	knifeCircumference					:LREAL :=857.65479443007;	(*[mm]*)
	startSyncAngle						:LREAL :=340.0;			(*[°]*)
	endSyncAngle						:LREAL :=20.0;			(*[°]*)
	startAngle							:LREAL :=90.0;			(*[°]*)
	stopAngle							:LREAL :=270.0;			(*[°]*)
	inflectionPoint						:LREAL :=50.0;			(*[%]*)
	numberOfKnives						:INT :=1;
	cutProfileCutOut						:DINT :=0;
	camProfilePhase1					:DINT :=0;
	jerkPhase1							:LREAL :=0.0;			(*[%]*)
	camProfilePhase2					:DINT :=0;
	jerkPhase2							:LREAL :=0.0;			(*[%]*)
	cutProfileCutIn						:DINT :=0;
	distanceToSensor					:LREAL :=0.0;			(*[mm]*)
	firstCutCorrection						:LREAL :=0.0;			(*[mm]*)
	startBacklashOffset					:LREAL :=50.0;			(*[mm]*)
	toStartPosVel						:LREAL :=10.0;			(*[mm/s]*)
	knifeOverspeedStartCut				:LREAL :=0.0;			(*[%]*)
	knifeOverspeedZero					:LREAL :=0.0;			(*[%]*)
	knifeOverspeedEndCut					:LREAL :=0.0;			(*[%]*)
	cpCorrectionMaximum					:LREAL :=0.0;			(*[mm]*)
	cpDeltaToleranceRangePositive			:LREAL :=0.0;			(*[mm]*)
	cpDeltaToleranceRangeNegative			:LREAL :=0.0;			(*[mm]*)
	adjustCutPositionPositiveValue			:LREAL :=0.0;			(*[mm]*)
	trimmCutPositionPositiveValue			:LREAL :=0.0;			(*[mm]*)
	adjustCutPositionNegativeValue			:LREAL :=0.0;			(*[mm]*)
	trimmCutPositionNegativeValue			:LREAL :=0.0;			(*[mm]*)
	cutPositionCorrectionVelocity			:LREAL :=0.0;			(*[mm/s]*)
	cutCorrWait						:INT :=0;
	shiftCorrectionStartPos					:LREAL :=0.0;			(*[%]percentageshiftinformatarea*)
	reStart							:BOOL :=FALSE;
	quickStart							:BOOL :=FALSE;
	formatlengthChangePossible				:BOOL :=FALSE;
	switchCAM							:BOOL :=FALSE;
	measuringEdge						:DINT :=0;
	cutPositionCorrectionOn				:BOOL :=FALSE;
	adjustCutPositionPositive				:BOOL :=FALSE;
	trimmCutPositionPositive				:BOOL :=FALSE;
	adjustCutPositionNegative				:BOOL :=FALSE;
	trimmCutPositionNegative				:BOOL :=FALSE;
	cleanCut							:BOOL :=FALSE;			(*cutwithoutcountingsheets*)
	torquePreControlOn					:BOOL :=FALSE;			(*activationoftorqueprecontrol*)
	totalInertiaOfRotaryKnifeSystem			:LREAL :=0.0;			(*[kgm²]totalinertiaofrotaryknifesystem*)
	torquePreControlMode					:DINT :=0;
	lookAHead							:LREAL :=0.0;			(*[µs]lookaheadtimeinCAM*)
	interruptProduction					:BOOL :=FALSE;
	continueProduction					:BOOL :=FALSE;
	leadingValueCouplingMode				:DINT :=0;
	syncLength							:LREAL :=0.0;			(*[mm]synchronizinglength*)
	extrapolationTime					:LREAL :=0.0;			(*[ms]extrapolationtimeonlyusedbyactualvaluecoupling*)
	constantVelocityAtCut					:BOOL :=FALSE;			(*=synchronousareawithconstantvirtualaxisvelocity,=synchronousareawithactualencodervelocity*)
	startLengthMode						:DINT :=0;
	startLength							:LREAL :=0.0;			(*[mm]*)
	stopLengthMode						:DINT :=0;
	stopLength							:LREAL :=0.0;			(*[mm]*)
	cuttingTorquePreControlOn				:BOOL :=FALSE;
	cuttingTorquePreControlActivePoints		:INT :=0;
	gearInRatioNumerator					:DINT :=0;
	gearInRatioDenominator				:DINT :=0;

END_STRUCT
END_TYPE

// ---- Library/AxisControl/DataTypes/TO_Cam_Struct_PointData.TcDUT
TYPE TO_Cam_Struct_PointData :
STRUCT
	x: LREAL;
	y:LREAL;

END_STRUCT
END_TYPE

// ---- Library/AxisControl/DataTypes/TO_Cam_Struct_SegmentData.TcDUT
TYPE TO_Cam_Struct_SegmentData :
STRUCT

	xmin:LREAL;
	xmax:LREAL;

	a0:LREAL;

	a1:LREAL;

	a2:LREAL;

	a3:LREAL;

	a4:LREAL;

	a5:LREAL;

	a6:LREAL;

	sineAmplitude:LREAL;

	sinePeriod:LREAL;

	sinePhase:LREAL;



END_STRUCT
END_TYPE

// ---- Library/Beckhoff/EL1008/DataTypes/EL1008_DEV_CONFIG.TcDUT
TYPE EL1008_DEV_CONFIG :
STRUCT
    // EN: Enables simulated input values for commissioning and diagnostics.
    // PT: Habilita valores simulados das entradas para comissionamento e diagnóstico.
    enableForce          : BOOL;
    forceDigitalInput_00 : BOOL;
    forceDigitalInput_01 : BOOL;
    forceDigitalInput_02 : BOOL;
    forceDigitalInput_03 : BOOL;
    forceDigitalInput_04 : BOOL;
    forceDigitalInput_05 : BOOL;
    forceDigitalInput_06 : BOOL;
    forceDigitalInput_07 : BOOL;
END_STRUCT
END_TYPE

// ---- Library/Beckhoff/EL1008/DataTypes/EL1008_HWTOPLC_PDOS.TcDUT
TYPE EL1008_HWTOPLC_PDOS :
STRUCT
    // EN: EL1008 EtherCAT input process data.
    // PT: Dados de processo das entradas EtherCAT do EL1008.
    digitalInput_00 AT %I* : BOOL;
    digitalInput_01 AT %I* : BOOL;
    digitalInput_02 AT %I* : BOOL;
    digitalInput_03 AT %I* : BOOL;
    digitalInput_04 AT %I* : BOOL;
    digitalInput_05 AT %I* : BOOL;
    digitalInput_06 AT %I* : BOOL;
    digitalInput_07 AT %I* : BOOL;
END_STRUCT
END_TYPE

// ---- Library/Beckhoff/EL1008/DataTypes/EL1008_PDOS.TcDUT
TYPE EL1008_PDOS :
STRUCT
    HwToPLC : EL1008_HWTOPLC_PDOS;
END_STRUCT
END_TYPE

// ---- Library/Beckhoff/EL1809/DataTypes/EL1809_DEV_CONFIG.TcDUT
TYPE EL1809_DEV_CONFIG :
    STRUCT
       
		enableForce	: BOOL;
		forceDigitalInput_00 : BOOL;
		forceDigitalInput_01 : BOOL;
		forceDigitalInput_02 : BOOL;
		forceDigitalInput_03 : BOOL;
		forceDigitalInput_04 : BOOL;
		forceDigitalInput_05 : BOOL;
		forceDigitalInput_06 : BOOL;
		forceDigitalInput_07 : BOOL;
		forceDigitalInput_08 : BOOL;
		forceDigitalInput_09 : BOOL;
		forceDigitalInput_10 : BOOL;
		forceDigitalInput_11 : BOOL;
		forceDigitalInput_12 : BOOL;
		forceDigitalInput_13 : BOOL;
		forceDigitalInput_14 : BOOL;
		forceDigitalInput_15 : BOOL;


    END_STRUCT
END_TYPE

// ---- Library/Beckhoff/EL1809/DataTypes/EL1809_HWTOPLC_PDOS.TcDUT
TYPE EL1809_HWTOPLC_PDOS :
	STRUCT
		
	
	digitalInput_00 AT %I* : BOOL;
	digitalInput_01 AT %I* : BOOL;
	digitalInput_02 AT %I* : BOOL;
	digitalInput_03 AT %I* : BOOL;
	digitalInput_04 AT %I* : BOOL;
	digitalInput_05 AT %I* : BOOL;
	digitalInput_06 AT %I* : BOOL;
	digitalInput_07 AT %I* : BOOL;
	digitalInput_08 AT %I* : BOOL;
	digitalInput_09 AT %I* : BOOL;
	digitalInput_10 AT %I* : BOOL;
	digitalInput_11 AT %I* : BOOL;
	digitalInput_12 AT %I* : BOOL;
	digitalInput_13 AT %I* : BOOL;
	digitalInput_14 AT %I* : BOOL;
	digitalInput_15 AT %I* : BOOL;


		
	END_STRUCT
END_TYPE

// ---- Library/Beckhoff/EL1809/DataTypes/EL1809_PDOS.TcDUT
TYPE EL1809_PDOS :
	STRUCT
		
		HwToPLC : EL1809_HWTOPLC_PDOS;
		
	END_STRUCT
END_TYPE

// ---- Library/Beckhoff/EL2809/DataTypes/EL2809_DEV_CONFIG.TcDUT
TYPE EL2809_DEV_CONFIG :
    STRUCT
       
		enableForce	: BOOL;
		forceDigitalOutput_00 : BOOL;
		forceDigitalOutput_01 : BOOL;
		forceDigitalOutput_02 : BOOL;
		forceDigitalOutput_03 : BOOL;
		forceDigitalOutput_04 : BOOL;
		forceDigitalOutput_05 : BOOL;
		forceDigitalOutput_06 : BOOL;
		forceDigitalOutput_07 : BOOL;
		forceDigitalOutput_08 : BOOL;
		forceDigitalOutput_09 : BOOL;
		forceDigitalOutput_10 : BOOL;
		forceDigitalOutput_11 : BOOL;
		forceDigitalOutput_12 : BOOL;
		forceDigitalOutput_13 : BOOL;
		forceDigitalOutput_14 : BOOL;
		forceDigitalOutput_15 : BOOL;
			


    END_STRUCT
END_TYPE

// ---- Library/Beckhoff/EL2809/DataTypes/EL2809_PDOS.TcDUT
TYPE EL2809_PDOS :
	STRUCT
		
		PlcToHw : EL2809_PLCTOHW_PDOS;
		
	END_STRUCT
END_TYPE

// ---- Library/Beckhoff/EL2809/DataTypes/EL2809_PLCTOHW_PDOS.TcDUT
TYPE EL2809_PLCTOHW_PDOS :
	STRUCT
		
		digitalOutput_00 AT %Q* : BOOL;
		digitalOutput_01 AT %Q* : BOOL;
		digitalOutput_02 AT %Q* : BOOL;
		digitalOutput_03 AT %Q* : BOOL;
		digitalOutput_04 AT %Q* : BOOL;
		digitalOutput_05 AT %Q* : BOOL;
		digitalOutput_06 AT %Q* : BOOL;
		digitalOutput_07 AT %Q* : BOOL;
		digitalOutput_08 AT %Q* : BOOL;
		digitalOutput_09 AT %Q* : BOOL;
		digitalOutput_10 AT %Q* : BOOL;
		digitalOutput_11 AT %Q* : BOOL;
		digitalOutput_12 AT %Q* : BOOL;
		digitalOutput_13 AT %Q* : BOOL;
		digitalOutput_14 AT %Q* : BOOL;
		digitalOutput_15 AT %Q* : BOOL;

	END_STRUCT
END_TYPE

// ---- Library/Beckhoff/EL3002 - Ai 2 x 10V - 12bit/DataTypes/EL3002_CHANNEL.TcDUT
TYPE EL3002_CHANNEL :
	STRUCT
		
	
	Status 	AT %I* : EL3002_DEV_STATUS;
	Value 	AT %I* : INT;
	
	
	END_STRUCT
END_TYPE

// ---- Library/Beckhoff/EL3002 - Ai 2 x 10V - 12bit/DataTypes/EL3002_DEV_CONFIG.TcDUT
TYPE EL3002_DEV_CONFIG :
    STRUCT
   
        // Setpoint scaling
       	channel1InputLow        : REAL := -32767.0;   // Minimum input value for setpoint		
        channel1InputHigh       : REAL := 32767.0; // Maximum input value for setpoint
        channel1OutputLow       : REAL := -100.0; // Minimum output value for setpoint
        channel1OutputHigh      : REAL := 100.0; // Maximum output value for setpoint
        // Setpoint scaling
       	channe12InputLow        : REAL := -32767.0;   // Minimum input value for setpoint		
        channe12InputHigh       : REAL := 32767.0; // Maximum input value for setpoint
        channe12OutputLow       : REAL := -100.0; // Minimum output value for setpoint
        channe12OutputHigh      : REAL := 100.0; // Maximum output value for setpoint		

    END_STRUCT
END_TYPE

// ---- Library/Beckhoff/EL3002 - Ai 2 x 10V - 12bit/DataTypes/EL3002_DEV_STATUS.TcDUT
TYPE EL3002_DEV_STATUS :
    STRUCT
      
		Underrange : BOOL;
		Overrange : BOOL;
		Limit1 : BOOL;
		Limit2 : BOOL;
		Error : BOOL;
		TxPDOState : BOOL;
		TxPDOToggle : BOOL;
	
    END_STRUCT
END_TYPE

// ---- Library/Beckhoff/EL3002 - Ai 2 x 10V - 12bit/DataTypes/EL3002_HWTOPLC_PDOS.TcDUT
TYPE EL3002_HWTOPLC_PDOS :
	STRUCT
		
	
	Channel1 	AT %I* : EL3002_CHANNEL;
	Channel2 	AT %I* : EL3002_CHANNEL;



	END_STRUCT
END_TYPE

// ---- Library/Beckhoff/EL3002 - Ai 2 x 10V - 12bit/DataTypes/EL3002_PDOS.TcDUT
TYPE EL3002_PDOS :
	STRUCT
		
		HwToPLC : EL3002_HWTOPLC_PDOS;
		
	END_STRUCT
END_TYPE

// ---- Library/Beckhoff/EL4004 - AQ 4 x 0-10V/DataTypes/EL4004_DEV_CONFIG.TcDUT
TYPE EL4004_DEV_CONFIG :
    STRUCT
   
        // Setpoint scaling
       	channel1InputLow        : REAL := 0.0;   // Minimum input value for setpoint		
        channel1InputHigh       : REAL := 100.0; // Maximum input value for setpoint
        channel1OutputLow       : REAL := 0.0; // Minimum output value for setpoint
        channel1OutputHigh      : REAL := 32767.0; // Maximum output value for setpoint

        // Setpoint scaling
       	channel2InputLow        : REAL := 0.0;   // Minimum input value for setpoint		
        channel2InputHigh       : REAL := 100.0; // Maximum input value for setpoint
        channel2OutputLow       : REAL := 0.0; // Minimum output value for setpoint
        channel2OutputHigh      : REAL := 32767.0; // Maximum output value for setpoint

        // Setpoint scaling
       	channel3InputLow        : REAL := 0.0;   // Minimum input value for setpoint		
        channel3InputHigh       : REAL := 100.0; // Maximum input value for setpoint
        channel3OutputLow       : REAL := 0.0; // Minimum output value for setpoint
        channel3OutputHigh      : REAL := 32767.0; // Maximum output value for setpoint

        // Setpoint scaling
       	channel4InputLow        : REAL := 0.0;   // Minimum input value for setpoint		
        channel4InputHigh       : REAL := 100.0; // Maximum input value for setpoint
        channel4OutputLow       : REAL := 0.0; // Minimum output value for setpoint
        channel4OutputHigh      : REAL := 32767.0; // Maximum output value for setpoint


    END_STRUCT
END_TYPE

// ---- Library/Beckhoff/EL4004 - AQ 4 x 0-10V/DataTypes/EL4004_HWTOPLC_PDOS.TcDUT
TYPE EL4004_HWTOPLC_PDOS :
	STRUCT
		
	
	Channel1 	AT %Q* : INT;
	Channel2 	AT %Q* : INT;
	Channel3 	AT %Q* : INT;
	Channel4 	AT %Q* : INT;

	END_STRUCT
END_TYPE

// ---- Library/Beckhoff/EL4004 - AQ 4 x 0-10V/DataTypes/EL4004_PDOS.TcDUT
TYPE EL4004_PDOS :
	STRUCT
		
		HwToPLC : EL4004_HWTOPLC_PDOS;
		
	END_STRUCT
END_TYPE

// ---- Library/Beckhoff/EL5152 -2 x  Encoder Input/DataTypes/EL5152_CONTROL.TcDUT
TYPE EL5152_CONTROL :
STRUCT

		{attribute 'hide'}
		_reserved1 : BIT;
		{attribute 'hide'}
		_reserved2 : BIT;
		Set_counter : BIT;
		{attribute 'hide'}
		_reserved3 : BIT;
		{attribute 'hide'}
		_reserved4 : BIT;
		{attribute 'hide'}
		_reserved5 : BIT;
		{attribute 'hide'}
		_reserved6 : BIT;
		{attribute 'hide'}
		_reserved7 : BIT;
		{attribute 'hide'}
		_reserved8 : USINT;
		
END_STRUCT
END_TYPE

// ---- Library/Beckhoff/EL5152 -2 x  Encoder Input/DataTypes/EL5152_DEV_CONFIG.TcDUT
TYPE EL5152_DEV_CONFIG :
STRUCT

	// Encoder configuration
	encoderPulsePerRevolution	: INT := 2000;      // Number of pulses per revolution (PPR) from the encoder
	encoderScalingFactor	    : REAL := 0.18;      // Position increment per pulse (e.g., 360 mm / 2000 PPR = 0.18 mm/pulse)
	moduloPosition 				: LREAL := 360.0	; // Modulo position range, for example 360.0 

	// Speed calculation
	speedCalculationCycleTime	: TIME := T#300MS;     // Interval at which encoder speed is recalculated

	// Simulation mode
	startSimulation				: BOOL := FALSE;    // Enables encoder simulation mode
	simulatedSpeed				: REAL := 10.0;     // Simulated speed in meters per minute (MPM)

	// Manual position set
	setPosition					: BOOL;             // Trigger to manually set encoder position
	desiredPosition				: LREAL;            // Desired encoder position in millimeters

END_STRUCT
END_TYPE

// ---- Library/Beckhoff/EL5152 -2 x  Encoder Input/DataTypes/EL5152_HWTOPLC.TcDUT
TYPE EL5152_HWTOPLC :
	STRUCT
		
			channel1 : EL5152_HWTOPLC_PDOS;
			channel2 : EL5152_HWTOPLC_PDOS;

	END_STRUCT
END_TYPE

// ---- Library/Beckhoff/EL5152 -2 x  Encoder Input/DataTypes/EL5152_HWTOPLC_PDOS.TcDUT
TYPE EL5152_HWTOPLC_PDOS :
	STRUCT
	
	status												: EL5152_STATUS;	
		{attribute 'hide'}
	_reserved1                                          : UINT;

	CounterValue                              : UDINT; // Current encoder counter value

	END_STRUCT
END_TYPE

// ---- Library/Beckhoff/EL5152 -2 x  Encoder Input/DataTypes/EL5152_PLCTOHW.TcDUT
TYPE EL5152_PLCTOHW :
	STRUCT
		
			channel1 : EL5152_PLCTOHW_PDOS;
			channel2 : EL5152_PLCTOHW_PDOS;

	END_STRUCT
END_TYPE

// ---- Library/Beckhoff/EL5152 -2 x  Encoder Input/DataTypes/EL5152_PLCTOHW_PDOS.TcDUT
TYPE EL5152_PLCTOHW_PDOS :
	STRUCT
		
		control					 : EL5152_CONTROL;
		setCounterValue			 : UDINT; // Sets the encoder counter value
		
	END_STRUCT
END_TYPE

// ---- Library/Beckhoff/EL5152 -2 x  Encoder Input/DataTypes/EL5152_STATUS.TcDUT
TYPE EL5152_STATUS :
STRUCT

		{attribute 'hide'}
		_reserved1 : BIT;
		{attribute 'hide'}
		_reserved2 : BIT;
		Set_counter_done : BIT;
		{attribute 'hide'}
		_reserved3 : BIT;
		{attribute 'hide'}
		_reserved4 : BIT;
		{attribute 'hide'}
		_reserved5 : BIT;
		{attribute 'hide'}
		_reserved6 : BIT;
		Extrapolation_stall : BIT;
		Status_of_input_A : BIT;
		Status_of_input_B : BIT;
		{attribute 'hide'}
		_reserved7 : BIT;
		{attribute 'hide'}
		_reserved8 : BIT;
		{attribute 'hide'}
		_reserved9 : BIT;
		Sync_error : BIT;
		{attribute 'hide'}
		_reserved10 : BIT;
		TxPDO_Toggle : BIT;	

END_STRUCT
END_TYPE

// ---- Library/EL6910 - TwinSAFE PLC/EL6910_ESTOP.TcDUT
TYPE EL6910_ESTOP :
STRUCT
	
	diagnostics : EL6910_ESTOP_DIGNOSTICS;
	status	: EL6910_ESTOP_STATUS;	

END_STRUCT
END_TYPE

// ---- Library/EL6910 - TwinSAFE PLC/EL6910_ESTOP_DIGNOSTICS.TcDUT
TYPE EL6910_ESTOP_DIGNOSTICS :
STRUCT

 	discrepancyErrGroup1       : BOOL; // Discrepancy error input group 1 - BIT00
    discrepancyErrGroup2       : BOOL; // Discrepancy error input group 2 - BIT01
    discrepancyErrGroup3       : BOOL; // Discrepancy error input group 3 - BIT02
    discrepancyErrGroup4       : BOOL; // Discrepancy error input group 4 - BIT03

    edmMonitoringErr1          : BOOL; // EDM monitoring error EDM1 - BIT04
    edmMonitoringErr2          : BOOL; // EDM monitoring error EDM2 - BIT05

    discrepancyErrGroup1_Safe  : BOOL; // Discrepancy error input group 1 with "Safe Inputs after Disc Error" - BIT08
    discrepancyErrGroup2_Safe  : BOOL; // Discrepancy error input group 2 with "Safe Inputs after Disc Error" - BIT09
    discrepancyErrGroup3_Safe  : BOOL; // Discrepancy error input group 3 with "Safe Inputs after Disc Error" - BIT10
    discrepancyErrGroup4_Safe  : BOOL; // Discrepancy error input group 4 with "Safe Inputs after Disc Error" - BIT11

END_STRUCT
END_TYPE

// ---- Library/EL6910 - TwinSAFE PLC/EL6910_ESTOP_STATUS.TcDUT
TYPE EL6910_ESTOP_STATUS :
STRUCT
	
    estopState_RUN        : BOOL; // RUN state 
    estopState_STOP       : BOOL; // STOP state 
    estopState_SAFE       : BOOL; // SAFE state 
    estopState_ERROR      : BOOL; // ERROR state 
    estopState_RESET      : BOOL; // RESET state 
    estopState_START      : BOOL; // START state 
    estopState_DELAYOUT   : BOOL; // DELAYOUT state 
	
END_STRUCT
END_TYPE

// ---- Library/EL6910 - TwinSAFE PLC/EL6910_HWTOPLC_PDOS.TcDUT
TYPE EL6910_HWTOPLC_PDOS :
	STRUCT
			
	EStop1State AT %I* : USINT;
	EStop1Diag 	AT %I* : UINT;
	
	EStop2State AT %I* : USINT;
	EStop2Diag 	AT %I* : UINT;

	EStop3State AT %I* : USINT;
	EStop3Diag 	AT %I* : UINT;

	EStop4State AT %I* : USINT;
	EStop4Diag 	AT %I* : UINT;	
	
	END_STRUCT
END_TYPE

// ---- Library/EL6910 - TwinSAFE PLC/EL6910_PDOS.TcDUT
TYPE EL6910_PDOS :
STRUCT
	
	HwToPLC : EL6910_HWTOPLC_PDOS;
	PlcToHw : EL6910_PLCTOHW_PDOS;			

END_STRUCT
END_TYPE

// ---- Library/EL6910 - TwinSAFE PLC/EL6910_PLCTOHW_PDOS.TcDUT
TYPE EL6910_PLCTOHW_PDOS :
	STRUCT
		
		ErrorAcknowledgement AT %Q* : BOOL;
		safetyReset AT %Q* : BOOL;
	
		Run AT %Q* : BOOL;
		
	END_STRUCT
END_TYPE

// ---- Library/FAS/IO-Link/006B51 - IO-Link Master/DataTypes/_006B51_Channel_State.TcDUT
TYPE _006B51_Channel_State :
STRUCT
	
	inputPin4 	 			: BOOL;
	inputPin2  				: BOOL;
	deviceState  			: BOOL;
	
    state_PortInNoDigitalInput        : BOOL;
    state_PortInNcDigitalInput        : BOOL;
    state_PortInDigitalOutput         : BOOL;
    state_PortInIoLink                : BOOL;

    state_NoDeviceDetected            : BOOL;
    state_IoLinkCommunicationStatus   : BOOL;
    state_InvalidVendorId             : BOOL;
    state_InvalidDeviceId             : BOOL;
    state_InvalidSerialNumber         : BOOL;
    state_InvalidCycleTime            : BOOL;
    state_InvalidProcessDataInLength  : BOOL;
    state_InvalidProcessDataOutLength : BOOL;
    state_InvalidIoLinkVersion        : BOOL;
	
END_STRUCT
END_TYPE

// ---- Library/FAS/IO-Link/006B51 - IO-Link Master/DataTypes/_006B51_HWTOPLC_PDOS.TcDUT
TYPE _006B51_HWTOPLC_PDOS :
STRUCT
	
	inputPin4 	 			: BYTE;
	inputPin2  				: BYTE;
	deviceState  			: BYTE;
	
	ioLinkDeviceState_Port0 : USINT;
	ioLinkDeviceState_Port1 : USINT;
	ioLinkDeviceState_Port2 : USINT;
	ioLinkDeviceState_Port3 : USINT;
	ioLinkDeviceState_Port4 : USINT;
	ioLinkDeviceState_Port5 : USINT;
	ioLinkDeviceState_Port6 : USINT;
	ioLinkDeviceState_Port7 : USINT;
	
END_STRUCT
END_TYPE

// ---- Library/FAS/IO-Link/00BE31 - IP67 16Di or 16Do/DataTypes/_00BE31_HWTOPLC_PDOS.TcDUT
TYPE _00BE31_HWTOPLC_PDOS :
STRUCT
	
	inputByte_0 	 : BYTE;
	inputByte_1  : BYTE;

END_STRUCT
END_TYPE

// ---- Library/FAS/IO-Link/00BE31 - IP67 16Di or 16Do/DataTypes/_00BE31_PLCTOHW_PDOS.TcDUT
TYPE _00BE31_PLCTOHW_PDOS :
STRUCT
	
	outputByte_0 	 : BYTE;
	outputByte_1 	 : BYTE;

END_STRUCT
END_TYPE

// ---- Library/FAS/IO-Link/00BH11 - 16Di or 16Do/DataTypes/_00BH11_HWTOPLC_PDOS.TcDUT
TYPE _00BH11_HWTOPLC_PDOS :
STRUCT
	
	inputByte_0 	 : BYTE;
	inputByte_1  : BYTE;

END_STRUCT
END_TYPE

// ---- Library/FAS/IO-Link/00BH11 - 16Di or 16Do/DataTypes/_00BH11_PLCTOHW_PDOS.TcDUT
TYPE _00BH11_PLCTOHW_PDOS :
STRUCT
	
	outputByte_0 	 : BYTE;
	outputByte_1 	 : BYTE;

END_STRUCT
END_TYPE

// ---- Library/FAS/IO-Link/00BW12 - 16 Solenoid Island/DataTypes/_00BW12_PLCTOHW_PDOS.TcDUT
TYPE _00BW12_PLCTOHW_PDOS :
STRUCT
	
	outputByte_0 	 : BYTE;
	outputByte_1 	 : BYTE;
	outputByte_2 	 : BYTE;
	outputByte_3 	 : BYTE;
	outputByte_4 	 : BYTE;
	outputByte_5 	 : BYTE;
	
END_STRUCT
END_TYPE

// ---- Library/FAS/IO-Link/0AC001 - Analog Input/DataTypes/_0AC001_DEV_CONFIG.TcDUT
TYPE _0AC001_DEV_CONFIG :
STRUCT
	
    // Raw analog input scaling (16-bit: 0..65535)
    analogInputLow   : REAL := 0.0;       // Minimum raw input value
    analogInputHigh  : REAL := 65535.0;   // Maximum raw input value (2 bytes)

    // Engineering-unit output scaling
    analogOutputLow  : REAL := 0.0;       // Engineering value at minimum input
    analogOutputHigh : REAL := 100.0;     // Engineering value at maximum input

END_STRUCT
END_TYPE

// ---- Library/FAS/IO-Link/0AC001 - Analog Input/DataTypes/_0AC001_HWTOPLC_PDOS.TcDUT
TYPE _0AC001_HWTOPLC_PDOS :
STRUCT
	
	inputByte_0 	 : BYTE;
	inputByte_1 	 : BYTE;

END_STRUCT
END_TYPE

// ---- Library/Machine/DryEnd/AutomaticOrderChange/aocConfig_TypeStruct.TcDUT
TYPE aocConfig_TypeStruct :
STRUCT

	automaticOrderChangeSpeed			: REAL	:= 50.0;		(*Automatic order change double facer speed*)

	automaticOrderChangeSpeedMult		: REAL 	:= 2;			(*Automatic order change speed multiplier*)
	rotaryKnifeSpeedMult				: REAL	:= 1;			(*Rotary knife speed multiplier this speed is going to be used to increase the dryend speed*)
	slitterSpeedMult					: REAL	:= 1;			(*slitter speed multiplier this speed is going to be used to reduce the sliiter speed *)

	rampUpTimeSec						: REAL	:= 5.0;		(*Ramp velocity in unit/s, with which the output is changed from a lower value to a higher one.*)
	rampDownTimeSec						: REAL 	:= -5.0;		(*Ramp velocity in unit/s, with which the output is changed from a higher value to a lower one.*)

	aocTimeout							: TIME	:= T#1M;		(*Maximum time to execute the AOC*)
	stackerDischargeDelay				: TIME 	:= T#10S;		(*Small  amout of time that the system  waits after the rotary knife sensor is clear to discharge the stacker*)
	changeSheetLengthTime				: TIME := T#10S;

	
	slitterPaperPresenceDelay					: TIME := T#5S;	
	
	
	speedControlPulseONTime				: TIME := T#1S;
	speedControlPulseOFFTime				: TIME := T#1S;

	
	rotaryShearCutX1MaxTime				: TIME := T#30S;
	measuringWheelClearMaxTime			: TIME := T#30S;	
	slitterClearMaxTime					: TIME := T#30S;	
	rotaryKnifeClearMaxTime				: TIME := T#30S;
	
	

END_STRUCT
END_TYPE

// ---- Library/Machine/DryEnd/AutomaticOrderChange/aocHmiCommands_TypeStruct.TcDUT
TYPE aocHmiCommands_TypeStruct :
STRUCT
	
	aocExecute : BOOL;

END_STRUCT
END_TYPE

// ---- Library/Machine/DryEnd/AutomaticOrderChange/aocHmiStatus_TypeStruct.TcDUT
TYPE aocHmiStatus_TypeStruct :
STRUCT
	
	automaticOrderChangeStatus	: STRING;

END_STRUCT
END_TYPE

// ---- Library/Machine/DryEnd/AutomaticOrderChange/lineControlHmiCommands_TypeStruct.TcDUT
TYPE lineControlHmiCommands_TypeStruct :
STRUCT
	
	speedInc : BOOL;
	speedDec : BOOL;
	speedStop : BOOL;

END_STRUCT
END_TYPE

// ---- Library/Machine/DryEnd/Hmi/hmiAlarms_TypeStruct.TcDUT
TYPE hmiAlarms_TypeStruct :
STRUCT

	slitter : hmiAlarmsSlitter_TypeStruct;
	rotaryKnife : hmiAlarmsRotaryKnife_TypeStruct;
	lowerStacker	: hmiAlarmsSimpleStacker_TypeStruct;
	upperStacker	: hmiAlarmsComplexStacker_TypeStruct;

END_STRUCT
END_TYPE

// ---- Library/Machine/DryEnd/Hmi/hmiCommands_TypeStruct.TcDUT
TYPE hmiCommands_TypeStruct :
STRUCT
	
	orderControl	: orderHmiCommands_TypeStruct;
	lineControl		: lineControlHmiCommands_TypeStruct;	
	slitter1		: slitterCommands_TypeStruct;
	upperKnife		: rotaryKnifeCommands_TypeStruct;
	lowerKnife		: rotaryKnifeCommands_TypeStruct;	
	
	lowerStacker	: hmiCommandsSimpleStacker_TypeStruct;
	upperStacker	: hmiCommandsComplexStacker_TypeStruct;
	
END_STRUCT
END_TYPE

// ---- Library/Machine/DryEnd/Hmi/hmiStatus_TypeStruct.TcDUT
TYPE hmiStatus_TypeStruct :
STRUCT
	alarmActive : BOOL;
		arrKnifeRunningMetersForSharpening		: ARRAY [1..5] OF INT;	(*This array is used to reset the lifetime meters that the knife runs*)
		arrKnifeRunningMetersForLubfrication	: ARRAY [1..5] OF INT;	(*This array is used to reset the lifetime meters that the knife runs*)
		slitter1 : slitterStatus_TypeStruct;
		
		upperKnife								: rotaryKnifeHmiStatus_TypeStruct;
		lowerKnife								: rotaryKnifeHmiStatus_TypeStruct;	
		machineMetrics 							: orderHmiStatus_TypeStruct;
		lowerStacker	: hmiStatusSimpleStacker_TypeStruct;
		upperStacker	: hmiStatusComplexStacker_TypeStruct;

		
END_STRUCT
END_TYPE

// ---- Library/Machine/DryEnd/Hmi/machineConfig_TypeStruct.TcDUT
TYPE machineConfig_TypeStruct :
STRUCT
	
	slitter1 : slitterConfig_TypeStruct;
	upperKnife : rotaryKnifeConfig_TypeStruct;
	lowerKnife	: rotaryKnifeConfig_TypeStruct;	
	automaticOrderChange : aocConfig_TypeStruct;	
	lowerStacker	: SimpleStackerConfig_TypeStruct;
	upperStacker	: ComplexStackerConfig_TypeStruct;

END_STRUCT
END_TYPE

// ---- Library/Machine/DryEnd/Order control/DataTypes/generatedOrderStatusWord_TypeStruct.TcDUT
TYPE generatedOrderStatusWord_TypeStruct :
STRUCT
	

	knifeOutOfRangeArr			: ARRAY [1..5] OF BOOL;
	scorerOutOfRangeArr		: ARRAY [1..8] OF BOOL;


	orderNotOk				: BOOL;	


END_STRUCT
END_TYPE

// ---- Library/Machine/DryEnd/Order control/DataTypes/generatedOrder_TypeStruct.TcDUT
TYPE generatedOrder_TypeStruct :
	STRUCT
		// ========================================================================
		// TOOLING SUMMARY
		// ========================================================================
		numberOfKnifes          : INT;              ///< Total count of active knives in this order
		numberOfScorers         : INT;              ///< Total count of active scorers in this order
		numberOfSheets          : INT;              ///< Total number of sheets in the current production list
		
		// ========================================================================
		// WEB GEOMETRY & CALCULATED WIDTHS [mm]
		// ========================================================================
		order1Width           : REAL;             ///< Calculated width of the Upper level order [mm]
		order2Width        	  : REAL;             ///< Calculated width of the Lower level order [mm]
		orderTotalWidth	      : REAL;             ///< Combined web width (Top + Bottom + Trim) [mm]
		firstKnifePosition      : REAL;             ///< Absolute position of the outermost left knife [mm]
		lastKnifePosition       : REAL;             ///< Absolute position of the outermost right knife [mm]
		
		// ========================================================================
		// KNIFE STATION DATA (Top/Rotary)
		// ========================================================================
		knifeEnabledArr         : ARRAY [1..10] OF BOOL; ///< Tool Enable: TRUE if knife index [x] is required
		knifePositionReferenceArr : ARRAY [1..10] OF REAL; ///< Target position for each knife [mm]
		
		// ========================================================================
		// SCORER STATION DATA (Creasing)
		// ========================================================================
		scorerEnabledArr        : ARRAY [1..20] OF BOOL; ///< Tool Enable: TRUE if scorer index [x] is required
		scorerPositionReferenceArr : ARRAY [1..20] OF REAL; ///< Target position for each scorer [mm]
		// ========================================================================
		// MACHINE STATUS
		// ========================================================================
		statusWord              : generatedOrderStatusWord_TypeStruct; ///< Structured status bits for order validity and errors
				

	END_STRUCT
END_TYPE
		// ========================================================================
		// MACHINE STATUS
		// ========================================================================
//		statusWord              : generatedOrderStatusWord_TypeStruct; ///< Structured status bits for order validity and errors

// ---- Library/Machine/DryEnd/Order control/DataTypes/orderConfig_TypeStruct.TcDUT
TYPE orderConfig_TypeStruct :
STRUCT
	

	automaticReduceMachineSpeed	: BOOL;		(*Reduce machine speed when order finishes*)
	autoStartAOC				: BOOL;		(*Start aoc automatic when the order finishes*)
	
	machineSpeedWhenOrderFinishes	: INT := 50;		(*Machine speed when the machine finishes the order*)
	
	orderFinishingAlertWhenRemainig	: INT := 100;		(*Used to alert the operator when the order is almost finished*)

	measuringWheelDiameter			: REAL := 264.3312;
	
END_STRUCT
END_TYPE

// ---- Library/Machine/DryEnd/Order control/DataTypes/orderHmiCommands_TypeStruct.TcDUT
TYPE orderHmiCommands_TypeStruct :
STRUCT
	
	changeOrder				: BOOL;
	resetUpperLevelCounter	: BOOL;	(*Reset upper level sheet counter*)
	resetLowerLevelCounter	: BOOL;	(*Reset lower level sheet counter*)

END_STRUCT
END_TYPE

// ---- Library/Machine/DryEnd/Order control/DataTypes/orderHmiStatus_TypeStruct.TcDUT
TYPE orderHmiStatus_TypeStruct :
STRUCT
	
	orderFinishing					: BOOL;
	orderFinished					: BOOL;
	linearMetersProduced			: DINT;
	arrMetersPerHour				: ARRAY [0..23] OF INT; (*Meters produced per hour*)
	arrMachineNotRunningTimePerHour	: ARRAY [0..23] OF INT; (*Machine stoped time per hour*)
	arrAverageSpeedPerHour			: ARRAY [0..23] OF INT; (*Machine average speed per hour*)
	machineNotRunningTimeTotal		: INT;
	
END_STRUCT
END_TYPE

// ---- Library/Machine/DryEnd/Order control/DataTypes/orderVariables_TypeStruct.TcDUT
TYPE orderVariables_TypeStruct :
STRUCT
    // ========================================================================
    // CUSTOMER & LOGISTICS DATA
    // ========================================================================
    id                      : DINT;             ///< Unique Order Identification Number
    product                 : STRING;           ///< Product name or internal SKU description
    client                  : STRING;           ///< Customer / Client name
    
    // ========================================================================
    // GEOMETRY & TOOLING CONFIGURATION
    // ========================================================================
    sheetType               : INT := 1;         ///< Scorer config: 0=None, 1=Two Scorers, 2=Four Scorers
    sheetQuantity           : INT := 2;         ///< Number of sheets/outs across the web width
    sheetLength             : INT := 1200;      ///< Cut-off length of each sheet [mm]
    
    // ========================================================================
    // SCORER / CREASER POSITIONS [mm]
    // ========================================================================
    sheetM1                 : INT := 100;       ///< Position of Scorer 1 [mm]
    sheetM2                 : INT := 100;       ///< Position of Scorer 2 [mm]
    sheetM3                 : INT := 100;       ///< Position of Scorer 3 [mm]
    sheetM4                 : INT := 0;         ///< Position of Scorer 4 [mm]
    sheetM5                 : INT := 0;         ///< Position of Scorer 5 [mm]
    
    // ========================================================================
    // PRODUCTION COUNTERS (CUTS)
    // ========================================================================
    numberOfCuts            : DINT;             ///< Total quantity of cuts required for order
    numberOfCutsProduced    : DINT;             ///< Successfully produced cut count
    numberOfCutsRemaining   : DINT;             ///< Calculated: (numberOfCuts - numberOfCutsProduced)
    
    // ========================================================================
    // STACKING & PILE MANAGEMENT
    // ========================================================================
    pileQuantity            : INT := 25;        ///< Target sheet count per finished stack (pile)
    pileQuantityProduced    : INT;              ///< Number of completed piles dispatched
    pileQuantityRemaining   : INT;              ///< Number of piles left to complete the order
    pileCounter             : INT;              ///< Current sheet count in the active pile (resets after pileQuantity)
    
    // ========================================================================
    // QUALITY & WASTE TRACKING
    // ========================================================================
    scrapCounter            : INT;              ///< Count of rejected or wasted sheets
   	counterReset			: BOOL;				///< Counter reset command
	
END_STRUCT
END_TYPE

// ---- Library/Machine/DryEnd/Order control/DataTypes/order_TypeStruct.TcDUT
TYPE order_TypeStruct :
STRUCT
    // ========================================================================
    // DATABASE & TRACKING LOGISTICS
    // ========================================================================
    startedAt               : STRING := '2026-01-11 13:07:00.000'; ///< Timestamp of order initiation
    tableID                 : DINT;                     ///< SQL Database Unique Index/Primary Key
    productionListNumber    : DINT := 92482;            ///< Production Planning System (ERP/MES) ID
    aocRequest      		: BOOL;                     ///< Trigger signal for order transition	
    changeOrderRequest      : BOOL;                     ///< Trigger signal for order transition
    saveSQLFinished         : BOOL;                     ///< Feedback: Database write operation successful
    saveSQLTimeOut          : BOOL;                     ///< Feedback: Database connection/write failure
   	plcWatchDog				: BOOL;
 
    // ========================================================================
    // BOARD SPECIFICATIONS (GRADE & COMPOSITION)
    // ========================================================================
    paperComposition        : STRING := 'KF3MF3K/BC 670G/M²'; ///< Board grade and total weight description
    fluteType               : STRING := 'BC';           ///< Corrugation profile (e.g., Single/Double Wall)
    paperWidth              : INT := 1810;              ///< Raw paper web width [mm]
    
    // ========================================================================
    // PAPER LAYER DEFINITIONS (LINERS & MEDIUMS)
    // ========================================================================
    paper1                  : STRING := 'KRAFT-90';     ///< Layer 1: Top Liner (Face)
    paper2                  : STRING := 'MIOLO F-130';  ///< Layer 2: Fluting 1 (Medium)
    paper3                  : STRING := 'MIOLO-90';     ///< Layer 3: Center Liner
    paper4                  : STRING := 'MIOLO-90';     ///< Layer 4: Fluting 2 (Medium)
    paper5                  : STRING := 'MIOLO-90';     ///< Layer 5: Bottom Liner (Back)
    
    // ========================================================================
    // PRODUCTION METRICS & KPI TRACKING
    // ========================================================================
    lineSpeed               : REAL;                     ///< Current machine velocity [m/min]
    linearMeters            : REAL := 2208.0;           ///< Total target length for the order [m]
    linearMetersProduced    : REAL;                     ///< Actual quantity processed [m]
    linearMetersRemaining   : REAL;                     ///< Calculated distance until completion [m]
    
    // ========================================================================
    // TOOLING & EXECUTION CONTROL
    // ========================================================================
    scorerHeightMM          : REAL := 0.5;              ///< Target penetration depth for slitter-scorer tools [mm]
    levelSelector           : E_LevelSelector := 1;     ///< Active Level: 1=Upper, 2=Lower, 3=Both
    invertOrderLevel        : BOOL;                     ///< Flag to swap logic between physical machine levels
    invertOrderSide         : BOOL;                     ///< Flag to swap order data between Order 1 and Order 2
 
    // ========================================================================
    // CHILD STRUCTURES (DETAILED PARAMETERS)
    // ========================================================================
    order1                  : OrderVariables_TypeStruct; ///< Config parameters for Upper Knife station
    order2                  : OrderVariables_TypeStruct; ///< Config parameters for Lower Knife station
    generatedOrder          : GeneratedOrder_TypeStruct; ///< Resultant set calculated for machine execution
    
END_STRUCT
END_TYPE

// ---- Library/Machine/DryEnd/Order control/DataTypes/sheetTypeEnum.TcDUT
(*
This enumerator is used to define the type of sheet that is going to be
produced by the machine
*)

TYPE sheetTypeEnum:
 (
	SHEET_WITH_NO_SCORER,		(* Sheet with no scoring marks*)
	SHEET_WITH_TWO_SCORER,		(* Sheet with two socoring marks *)
	SHEET_WITH_FOUR_SCORER		(*Sheet with four socoring marks*)

 );
END_TYPE

// ---- Library/Machine/Rotary knife/Config/rotaryKnifeConfig_TypeStruct.TcDUT
(*
TYPE rotaryKnifeConfig_TypeStruct :
STRUCT
	
	infeedRollSpeedOffset	: REAL	:= 1.1;
	outfeedRollSpeedOffset	: REAL	:= 1.2;
	minLineSpeed			: REAL := 20.0;
	
	switchEncoderDelay			: TIME := T#30S;
	speedCurve				    : ARRAY [1..10] OF rotaryKnifeSpeedCurve_TypeConfig;

	lengthAdjustment			: INT;
	
END_STRUCT
END_TYPE 
*)
TYPE rotaryKnifeConfig_TypeStruct :
STRUCT
    
    // --- Roll Speed Ratios ---
    infeedRollSpeedOffset   : REAL := 1.1;  // Multiplier for infeed roll speed relative to line speed (e.g., 1.1 = 10% draw)
    outfeedRollSpeedOffset  : REAL := 1.2;  // Multiplier for outfeed roll speed to maintain tension/gap after cut
    
    // --- Operational Limits ---
    minLineSpeed            : REAL := 20.0; // Minimum line speed (e.g., m/min) to allow automatic operation
    
    // --- Geometry & Logic ---
    enableSyncDiameter      : BOOL;         // TRUE: Use synchronous cutting if sheet length < Knife Circumference (π * D)
    knifeDiameter           : REAL := 262.670; // Physical diameter of the knife cylinder (mm)
    knifeDiameterFactor           	: REAL := 1.0; // Physical diameter of the knife cylinder (mm)
    
	
    // --- Timing & Profiles ---
    switchEncoderDelay      : TIME := T#30S; // Delay/filter time when toggling between feedback encoders
    speedCurve              : ARRAY [1..10] OF rotaryKnifeSpeedCurve_TypeConfig; // CAM or velocity profiles for different materials/speeds

    // --- Fine Tuning ---
    lengthAdjustment        : INT;          // Global position offset (pulses or tenths of mm) to trim cut accuracy
    
END_STRUCT
END_TYPE

// ---- Library/Machine/Rotary knife/Config/rotaryKnifeHmiStatus_TypeStruct.TcDUT
TYPE rotaryKnifeHmiStatus_TypeStruct :
STRUCT


	statusWord1 : rotaryKnifeStatusWord1_TypeStruct;
	statusWord2 : rotaryKnifeStatusWord2_TypeStruct;
	
	speedLimitActive	: BOOL;
	speedCurveActive	: INT;
	maxSpeed			: REAL;
	totalOfCuts	: DINT;
	sheetLength : REAL;
	

END_STRUCT
END_TYPE

// ---- Library/Machine/Rotary knife/Config/rotaryKnifeSpeedCurve_TypeConfig.TcDUT
TYPE rotaryKnifeSpeedCurve_TypeConfig :
STRUCT
	
	machineSpeed	: REAL := 150;
	sheetLength		: REAL	:= 800;

END_STRUCT
END_TYPE

// ---- Library/Machine/Rotary knife/Config/rotaryKnifeStatusWord1_TypeStruct.TcDUT
TYPE rotaryKnifeStatusWord1_TypeStruct :
STRUCT
	
   	knifeAtHomeParkPos1             : BOOL;
    homingInProgress                : BOOL;
    homingComplete                  : BOOL;
    knifeInspectionMotionInProgress : BOOL;
    knifeInspectionMotionComplete   : BOOL;
    returnHomeMotionInProgress      : BOOL;
    returnHomeMotionComplete        : BOOL;
    jogForwardInProgress            : BOOL;
    jogReverseInProgress            : BOOL;
    knifeGearingOut                 : BOOL;
    knifeRunningEngaged             : BOOL;
    knifeStoppedDisengaged          : BOOL;
    maxLineSpeedLimitCalculated     : BOOL;
    batchMaxLineSpeedCalcInProgress : BOOL;
    batchMaxLineSpeedCalculated     : BOOL;
    watchdogClockOut                : BOOL;

END_STRUCT
END_TYPE

// ---- Library/Machine/Rotary knife/Config/rotaryKnifeStatusWord2_TypeStruct.TcDUT
TYPE rotaryKnifeStatusWord2_TypeStruct :
STRUCT
	
    batchSingleShotStopInProgress   : BOOL;
    registrationMarkMissed          : BOOL;
    registrationWindowOpen          : BOOL;
    registrationMarkAccepted        : BOOL;
    onLastBatch                     : BOOL;
    onLastCutOfLastBatch            : BOOL;
    pls1Output                      : BOOL;
    pls2Output                      : BOOL;
    referenceEnabled                : BOOL;
    driveHealthy                    : BOOL;
    reserved10                      : BOOL;
    reserved11                      : BOOL;
    userDefinedStatusBit12          : BOOL;
    userDefinedStatusBit13          : BOOL;
    userDefinedStatusBit14          : BOOL;
    userDefinedStatusBit15          : BOOL;

END_STRUCT
END_TYPE

// ---- Library/Machine/Rotary knife/Hmi/hmiAlarmsRotaryKnife_TypeStruct.TcDUT
TYPE hmiAlarmsRotaryKnife_TypeStruct :
STRUCT
    // Rotary Knife Specific Alarms
    exitGuardOpen                   : BOOL; // Alarm active - Exit guard open
    infeedGuardOpen                 : BOOL; // Alarm active - Infeed guard open
    exhaustDepressurized            : BOOL; // Alarm active - Exhaust system depressurized
    upperKnifeGuardClosed           : BOOL; // Alarm active - Upper knife guard open (Low Active)
    upperKnifeOilLevelLow           : BOOL; // Alarm active - Upper knife oil level low
    upperKnifeJamDetected           : BOOL; // Alarm active - Upper knife jam detected
    upperKnifeInfeedDrvOK           : BOOL; // Alarm active - Upper knife infeed drive fault (Low Active)
    upperKnifeOutfeedDrvOK          : BOOL; // Alarm active - Upper knife outfeed drive fault (Low Active)
    upperKnifeMainDrvOK             : BOOL; // Alarm active - Upper knife main drive fault (Low Active)
    upperKnifeSlave1DrvOK           : BOOL; // Alarm active - Upper knife slave 1 drive fault (Low Active)
    upperKnifeSlave2DrvOK           : BOOL; // Alarm active - Upper knife slave 2 drive fault (Low Active)
	upperKnifeNotActive				: BOOL;
	upperKnifeCutDisabled			: BOOL;

    
	lowerKnifeGuardClosed           : BOOL; // Alarm active - Lower knife guard open (Low Active)
    lowerKnifeOilLevelLow           : BOOL; // Alarm active - Lower knife oil level low
    lowerKnifeJamDetected           : BOOL; // Alarm active - Lower knife jam detected
    lowerKnifeInfeedDrvOK           : BOOL; // Alarm active - Lower knife infeed drive fault (Low Active)
    lowerKnifeOutfeedDrvOK          : BOOL; // Alarm active - Lower knife outfeed drive fault (Low Active)
    lowerKnifeMainDrvOK             : BOOL; // Alarm active - Lower knife main drive fault (Low Active)
    lowerKnifeSlave1DrvOK           : BOOL; // Alarm active - Lower knife slave 1 drive fault (Low Active)
    lowerKnifeSlave2DrvOK           : BOOL; // Alarm active - Lower knife slave 2 drive fault (Low Active)
	lowerKnifeNotActive				: BOOL;
	lowerKnifeCutDisabled			: BOOL;
	
END_STRUCT
END_TYPE

// ---- Library/Machine/Rotary knife/Hmi/rotaryKnifeCommands_TypeStruct.TcDUT
TYPE rotaryKnifeCommands_TypeStruct :
STRUCT

   	powerONCmd            : BOOL;
    powerOFFCmd           : BOOL;
  	jogFwCmd              : BOOL;
    jogRevCmd             : BOOL;
    cutCmd                : BOOL;
 
	resetTotalOfCuts	 :BOOL;
	
END_STRUCT
END_TYPE

// ---- Library/Machine/Rotary knife/Hmi/rotaryKnifeStatus_TypeStruct.TcDUT
TYPE rotaryKnifeStatus_TypeStruct :
	STRUCT
	
		lowerLevelSpeedRPM	: INT;
		lowerLevelKnifeSpeedMPM	: INT;
	
		lowerLevelMotorCurrent	: INT;
		
		lowerLevelInfeedSpeedRPM	: INT;
		lowerLevelInfeedEncoderMPM	: INT;
		lowerLevelInfeedMotorCurrent	: INT;
		
		lowerLevelOutfeedSpeedRPM	: INT;
		lowerLevelOutfeeddEncoderMPM	: INT;
		lowerLevelOutfeedMotorCurrent	: INT;
		
		
		upperLevelKnifeSpeedMPM	: INT;
		upperLevelEncoderMPM	: INT;
		upperLevelMotorCurrent	: INT;
		
		upperLevelInfeedSpeedRPM	: INT;
		upperLevelInfeedEncoderMPM	: INT;
		upperLevelInfeedMotorCurrent	: INT;
		
		upperLevelOutfeeddEncoderMPM	: INT;
		upperLevelOutfeedMotorCurrent	: INT;
		
		
	END_STRUCT
END_TYPE

// ---- Library/Machine/Slitter/DataTypes/Hmi/E_LevelSelector.TcDUT
{attribute 'qualified_only'}
TYPE E_LevelSelector : (
	
    eUpperOnly := 1,   // Only upper level enabled
    eLowerOnly := 2,   // Only lower level enabled
    eBoth      := 3    // Upper + Lower enabled
);
END_TYPE

// ---- Library/Machine/Slitter/DataTypes/Hmi/hmiAlarmsSlitter_TypeStruct.TcDUT
TYPE hmiAlarmsSlitter_TypeStruct :
STRUCT
	

	safetyCircuitFault								: BOOL;
	slitterHomeNotCompleteFault							: BOOL;
	slitterTractionNotEnabledFault					: BOOL;
	
	knife01Fault								: BOOL;
	knife02Fault								: BOOL;
	knife03Fault								: BOOL;
	knife04Fault								: BOOL;
	knife05Fault								: BOOL;
	knife06Fault								: BOOL;
	knife07Fault								: BOOL;
	

	upperScorer01Fault								: BOOL;
	upperScorer02Fault								: BOOL;
	upperScorer03Fault								: BOOL;
	upperScorer04Fault								: BOOL;
	upperScorer05Fault								: BOOL;
	upperScorer06Fault								: BOOL;
	upperScorer07Fault								: BOOL;
	upperScorer08Fault								: BOOL;
	upperScorer09Fault								: BOOL;
	upperScorer10Fault								: BOOL;
	upperScorer11Fault								: BOOL;
	upperScorer12Fault								: BOOL;
	
	

	lowerScorer01Fault								: BOOL;
	lowerScorer02Fault								: BOOL;
	lowerScorer03Fault								: BOOL;
	lowerScorer04Fault								: BOOL;
	lowerScorer05Fault								: BOOL;
	lowerScorer06Fault								: BOOL;
	lowerScorer07Fault								: BOOL;
	lowerScorer08Fault								: BOOL;
	lowerScorer09Fault								: BOOL;
	lowerScorer10Fault								: BOOL;
	lowerScorer11Fault								: BOOL;
	lowerScorer12Fault								: BOOL;
	
	
	orderFault			:BOOL;

	knife1OutOfRange	:BOOL;
	knife2OutOfRange	:BOOL;
	knife3OutOfRange	:BOOL;
	knife4OutOfRange	:BOOL;
	knife5OutOfRange	:BOOL;
	
	scorer1OutOfRange	:BOOL;
	scorer2OutOfRange	:BOOL;
	scorer3OutOfRange	:BOOL;
	scorer4OutOfRange	:BOOL;
	scorer5OutOfRange	:BOOL;
	scorer6OutOfRange	:BOOL;
	scorer7OutOfRange	:BOOL;
	scorer8OutOfRange	:BOOL;
	
	
	
	
	

    // Scorer traction (main traction axis for scorers)
    scorerTractionFault          : BOOL;
	knifeTractionFault : BOOL;	
    // ─────────────── SCORER HEIGHT ───────────────
    scorerHeightAxisFault        : BOOL;

    // ─────────────── SCRAP TRIMMING ───────────────
    scrapTrimOperatorSideFault   : BOOL;
    scrapTrimDriveSideFault      : BOOL;
END_STRUCT
END_TYPE

// ---- Library/Machine/Slitter/DataTypes/Hmi/hmiCommandsFlaps_TypeStruct.TcDUT
TYPE hmiCommandsFlaps_TypeStruct :
STRUCT
		
	upCmd	 :BOOL;
	downCmd	: BOOL;

END_STRUCT
END_TYPE

// ---- Library/Machine/Slitter/DataTypes/Hmi/hmiCommandsJog_TypeStruct.TcDUT
TYPE hmiCommandsJog_TypeStruct :
STRUCT
		
	jogFw	 :BOOL;
	jogRev	: BOOL;

END_STRUCT
END_TYPE

// ---- Library/Machine/Slitter/DataTypes/Hmi/hmiCommandsSmallPosCorrection_TypeStruct.TcDUT
TYPE hmiCommandsSmallPosCorrection_TypeStruct :
STRUCT
	
	positionCorrection	: REAL;
	execute				: BOOL;

END_STRUCT
END_TYPE

// ---- Library/Machine/Slitter/DataTypes/Hmi/hmiSlitterAlarms_TypeStruct.TcDUT
TYPE hmiSlitterAlarms_TypeStruct :
STRUCT
	
	(*Circuit Breaker Fault*)
	(*_________________________________________________*)	
	knifeRobotCircuitBreaker		: BOOL;
	innerScorerRobotCircuitBreaker	: BOOL;
	outerScorerRobotCircuitBreaker	: BOOL;
	knifeTractionCircuitBreaker		: BOOL;
	scorerTractionCircuitBreaker	: BOOL;
	trimSuctionCircuitBreaker		: BOOL;
	
	(*Drive Fault*)
	(*_________________________________________________*)
	knifeRobotFault					: BOOL;
	innerScorerRobotFault			: BOOL;
	outerScorerRobotFault			: BOOL;
	knifeTractionFault				: BOOL;
	scorerTractionFault				: BOOL;
	
	(*Ethercat fault*)
	(*_________________________________________________*)
	ioLinkMasterEthercatFault		: BOOL;
	knifeRobotEthercatFault			: BOOL;
	innerScorerRobotEthercatFault	: BOOL;
	outerScorerRobotEthercatFault	: BOOL;
	knifeTractionEthercatFault		: BOOL;
	scorerTractionEthercatFault		: BOOL;
	
	(*IO-Link Fault*)
	(*_________________________________________________*)	
	ioLinkPort0Fault				: BOOL;
	ioLinkPort1Fault				: BOOL;
	ioLinkPort2Fault				: BOOL;
	ioLinkPort3Fault				: BOOL;
	ioLinkPort4Fault				: BOOL;
	ioLinkPort5Fault				: BOOL;
	ioLinkPort6Fault				: BOOL;
	ioLinkPort7Fault				: BOOL;
	
	(*Process fault*)	
	(*_________________________________________________*)
	(*Knife*)
	knifeRobotNotHomed						: BOOL;
	knifeRobotLimOP							: BOOL;
	knifeRobotLimST							: BOOL;
	knifeToolLimOP							: BOOL;
	knifeToolLimST							: BOOL;
	knifeNotFound							: BOOL;
	knifePositionSetpointOutOfRange			: BOOL;
	knifePositionLagExceeded				: BOOL;
	
	
	(*Inner scorer fault*)
	innerScorerRobotNotHomed				: BOOL;
	innerScorerRobotLimOP					: BOOL;
	innerScorerRobotLimST					: BOOL;
	innerScorerToolLimOP					: BOOL;
	innerScorerToolLimST					: BOOL;
	innerScorerNotFound						: BOOL;
	innerScorerPositionSetpointOutOfRange	: BOOL;
	innerScorerPositionLagExceeded			: BOOL;


	
	(*Outer scorer fault*)
	outerScorerRobotNotHomed				: BOOL;
	outerScorerRobotLimOP					: BOOL;
	outerScorerRobotLimST					: BOOL;
	outerScorerToolLimOP					: BOOL;
	outerScorerToolLimST					: BOOL;
	outerScorerNotFound						: BOOL;
	outerScorerPositionSetpointOutOfRange	: BOOL;
	outerScorerPositionLagExceeded			: BOOL;



	
	(*Safety fault*)
	(*_________________________________________________*)	
	safetyRelayNotOK						: BOOL;
	
	
	(*General faults*)
	
	notPossibleToExecutePositioning			: BOOL;		(*Not possible to execute automatic positioning while machine is in manual*)
	generatedOrderError						: BOOL;
	
	
	
	

END_STRUCT
END_TYPE

// ---- Library/Machine/Slitter/DataTypes/Hmi/slitterCommands_TypeStruct.TcDUT
TYPE slitterCommands_TypeStruct :
STRUCT

	tractionMotorAutoMan			: BOOL;	(*Knife / scorer motor automatic manual (0 = Auto / 1 = Manual)*)
	tractionMotorSpeed				: INT;		(*Traction motor manual speed reference in meters per minute*)
	knifeMotorRun					: BOOL;	(*Start / Stop knife motor*)
	scorerMotorRun					: BOOL;	(*Start / Stop scorer motor*)
	enablePositioningAxis			: BOOL;	(*Enable positioning axis*)
	executeHomming					: BOOL;	(*Execute homming*)
	enableAxis						: BOOL;	(*Enable positioning axis*)
	executePositioning				: BOOL;	(*Execute positioning*)

	resetCommand					: BOOL;	(**)

	startCutting					: BOOL;	(*Start / Stop cutting*)
	generatePositions				: BOOL;	(*Generate order positions*)
	changeOrder						: BOOL;	(*Change order*)

	paperTrimSuctionOpen			: BOOL;	(*Paper trim suction motor open*)
	paperTrimSuctionClose			: BOOL;	(*Paper trim suction motor close*)
	paperTrimSuctionAutoPos			: BOOL;	(*Paper trim suction motor automatic positioning*)
	paperTrimSuctionHome			: BOOL;	(*Paper trim suction motor home*)
	paperTrimSuctionPosSetpoint		: INT;	(*Paper trim suction motor position setpoint*)

	scorerHeightIncrement			: BOOL;	(*Scorer height increment*)
	scorerHeightDecrement			: BOOL;	(*Scorer height decrement*)
	scorerHeightHome				: BOOL;	(*Scorer height execute home*)
	scorerHightPos					: BOOL;	(*Scorer height execute positioning*)
	scorerHeightAutoMan				: BOOL;	(*Scorer height auto / manual (0 = Auto / 1 = Manual)*)

	autoManualCommand				: BOOL;	(*Slitter automatic / manual positioning*)
	moveKnifeOpSide					: BOOL;
	moveKnifeStSide					: BOOL;
	searchKnifeManual				: BOOL;

	moveInnerScorerOpSide			: BOOL;
	moveInnerScorerStSide			: BOOL;
	searchInnerScorerManual			: BOOL;


	moveOuterScorerOpSide			: BOOL;
	moveOuterScorerStSide			: BOOL;
	searchOuterScorerManual			: BOOL;

	moveMachineOperatorSide			: BOOL;	(*Move slitter to operator side*)
	moveMachineSteamSide			: BOOL;	(*Move slitter to steam side*)


	knifeRunningMetersResetArr		: ARRAY [1..20] OF BOOL;	(*This array is used to reset the lifetime meters that the knife runs*)
	knifeManualSharpeningArr		: ARRAY [1..20] OF BOOL;	(*This array is used to sharpen the knife manualy*)
	knifeManualLubrificationArr		: ARRAY [1..20] OF BOOL;	(*This array is used to lubrificate the knife manualy*)
	knifeEnabledArr					: ARRAY [1..20] OF BOOL;	(*Tool enabled array*)
	scorerEnabledArr				: ARRAY [1..20] OF BOOL;	(*Tool enabled array*)
	scorerSolenoidArr				: ARRAY [1..20] OF BOOL;	(*Tool positions*)
	knifeSolenoidArr				: ARRAY [1..20] OF BOOL;	(*Tool positions*)
	
	
	knifeJogArr						: ARRAY [1..5] OF hmiCommandsJog_TypeStruct;
	scorerJogArr						: ARRAY [1..8] OF hmiCommandsJog_TypeStruct;
	knifePosCorrectionArr				: ARRAY [1..5] OF hmiCommandsSmallPosCorrection_TypeStruct;
	scorerPosCorrectionArr				: ARRAY [1..8] OF hmiCommandsSmallPosCorrection_TypeStruct;

    // ─────────────── KNIFE MAINTENANCE (HMI COMMANDS) ───────────────
    knifeManualSharpeningCmdArr       : ARRAY [1..20] OF BOOL; // Manual knife sharpening command (per knife) / Comando manual de afiação (por faca)
    knifeManualLubrificationCmdArr    : ARRAY [1..20] OF BOOL; // Manual knife lubrication command (per knife) / Comando manual de lubrificação (por faca)

	
    // ─────────────── FLAPS / DIVERTERS ───────────────
    flapsAllUP                    : BOOL;  // TRUE when all flaps are in UP position / TRUE quando todas as aletas estão para cima
    flapsAllDown                  : BOOL;  // TRUE when all flaps are in DOWN position / TRUE quando todas as aletas estão para baixo
    flapsSetAuto                  : BOOL;  // Flap system in automatic mode / Sistema de aletas em automático
	flapsInvertDirection		  : BOOL;
	
    flapsManualCmdArr             : ARRAY [1..27] OF hmiCommandsFlaps_TypeStruct;  // Manual commands per flap / Comandos manuais por alet
	
	
    // ─────────────── GENERAL / SEQUENCES ───────────────
    resetCmd                      : BOOL;  // Reset commands, states and latched faults / Reset de comandos, estados e falhas

    enableAxisCmd                 : BOOL;  // Enable slitter positioning axes (power/permit motion) / Habilita eixos de posicionamento
    disableAxisCmd                : BOOL;  // Disable slitter positioning axes / Desabilita eixos de posicionamento

    executePositioningCmd         : BOOL;  // Start positioning sequence (pulse/edge) / Executa sequência de posicionamento (pulso)
    executePosCorrectionCmd       : BOOL;  // Start position correction routine (pulse/edge) / Executa correção de posição (pulso)
    executeHomeCmd                : BOOL;  // Start homing sequence (pulse/edge) / Executa homing (pulso)

    // ─────────────── TRACTION MOTOR ───────────────
    tractionMotorStartCmd         : BOOL;  // Start command for slitter traction motor / Partida motor de tração do slitter
    tractionMotorStopCmd          : BOOL;  // Stop command for slitter traction motor / Parada motor de tração do slitter

    // ─────────────── SLITTER CARRIAGE MANUAL MOVE ───────────────
    moveSlitterOperatorSideCmd    : BOOL;  // Slitter carriage move OS / Movimento carro slitter LO (lado operador)
    moveSlitterDriveSideCmd       : BOOL;  // Slitter carriage move DS / Movimento carro slitter LA (lado acionamento)

    // ─────────────── SCORER HEIGHT CONTROL ───────────────
    scorerHeightIncCmd            : BOOL;  // Increase scorer height / Sobe altura do scorer
    scorerHeightDecCmd            : BOOL;  // Decrease scorer height / Desce altura do scorer

    scorerHightPosCmd             : BOOL;  // Execute scorer height positioning / Executa posicionamento da altura do scorer

    // ─────────────── TRIM DUCT LIMIT SENSORS (COMMAND/STATUS) ───────────────
    osTrimDuctSensorOpenCmd       : BOOL;  // OS trim duct sensor — maximum limit reached / Sensor duto refilo LO — limite máximo atingido
    osTrimDuctSensorCloseCmd      : BOOL;  // OS trim duct sensor — minimum limit reached / Sensor duto refilo LO — limite mínimo atingido

    dsTrimDuctSensorOpenCmd       : BOOL;  // DS trim duct sensor — maximum limit reached / Sensor duto refilo LA — limite máximo atingido
    dsTrimDuctSensorCloseCmd      : BOOL;  // DS trim duct sensor — minimum limit reached / Sensor duto refilo LA — limite mínimo atingido

    // ─────────────── OUTFEED ROLLS COMMAND ───────────────
	
  	outfeedRoll_ManCmd      : BOOL; // Manual Mode activation command
    outfeedRoll_UpCmd       : BOOL; // Manual command to raise the roll
    outfeedRoll_DownCmd     : BOOL; // Manual command to lower the roll
	


    // ─────────────── JOG COMMANDS ───────────────
    knifeJogCmdArr                : ARRAY [1..7] OF hmiCommandsJog_TypeStruct;   // Knife jog commands (per knife) / Jog das facas (por faca)
    scorerJogCmdArr               : ARRAY [1..12] OF hmiCommandsJog_TypeStruct;  // Scorer jog commands (per scorer) / Jog dos scorers (por scorer)


END_STRUCT
END_TYPE

// ---- Library/Machine/Slitter/DataTypes/Hmi/slitterConfig_TypeStruct.TcDUT
TYPE slitterConfig_TypeStruct :
STRUCT
    // ------------------------------------------------------------
    // Machine
    // ------------------------------------------------------------
    machineWidth            : INT := 2200;   (* Machine total width *)
    machineNumberOfKnifes   : INT := 5;      (* Machine number of knifes *)
    machineNumberOfScorers  : INT := 8;      (* Machine number of scorers *)

    // ------------------------------------------------------------
    // Home positions
    // (based on the values shown in the screenshots)
    // ------------------------------------------------------------
    homePositionKnife  : ARRAY [1..5] OF REAL := [184, 330, 477, 1907, 2060];
    homePositionScorer : ARRAY [1..8] OF REAL := [204, 202, 364, 340, 1864, 1890, 2004, 2050];

    // ------------------------------------------------------------
    // Homing
    // ------------------------------------------------------------
    toolHommingVelocity     : LREAL := 50;
    toolHommingAccel        : LREAL := 242.682;
    toolHommingDecel        : LREAL := 242.682;
    toolHommingTimeLimit    : DINT  := 9999; (* Homming time limit in seconds *)

    // ------------------------------------------------------------
    // Parking
    // ------------------------------------------------------------
    toolParkingPosition     : LREAL := 40;

    // ------------------------------------------------------------
    // Tool search profile
    // ------------------------------------------------------------
    toolSearchVelocity      : LREAL := 150;       (* Tool search velocity *)
    toolSearchAccel         : LREAL := 242.682;   (* Tool acceleration *)
    toolSearchDecel         : LREAL := 970.726;   (* Tool deceleration *)
    toolSearchJerk          : LREAL := 89486.1;   (* Tool search jerk *)

    // ------------------------------------------------------------
    // Positioning profiles
    // ------------------------------------------------------------
    toolFastPositioningVelocity : LREAL := 180;
    toolFastPositioningAccel    : LREAL := 242.682;
    toolFastPositioningDecel    : LREAL := 180;
    toolFastPositioningJerk     : LREAL := 5592.86;

    toolSlowPositioningVelocity : LREAL := 40;
    toolSlowPositioningAccel    : LREAL := 200;
    toolSlowPositioningDecel    : LREAL := 900;
    toolSlowPositioningJerk     : LREAL := 5592.86;

    // ------------------------------------------------------------
    // General / Manual motion
    // ------------------------------------------------------------
    toolGeneralMotionVelocity    : LREAL := 100;
    toolGeneralMotionAccel       : LREAL := 242.682;
    toolGeneralMotionDecel       : LREAL := 242.682;
    toolGeneralMotionJerk        : LREAL := 5592.86;

    toolManualMotionVelocity     : LREAL := 80;
    toolManualMotionAccel        : LREAL := 242.682;
    toolManualMotionDecel        : LREAL := 242.682;
    toolManualMotionJerk         : LREAL := 5592.86;

    // ------------------------------------------------------------
    // Maintenance counters
    // ------------------------------------------------------------
    knifeSharpeningTime      : INT := 10000;  (* Knife sharpening time in seconds *)
    knifeSharpeningDistance  : INT := 250;    (* Knife sharpening distance in meters *)

    knifeLubrificationTime   : INT := 500;    (* Knife lubrification time in seconds *)
    knifeLubrificationDistance : INT := 1000; (* Knife lubrification distance in meters *)

    //=================================================================
    // KNIFE AUXILIARY FUNCTIONS (SHARPENING / LUBRICATION)
    //=================================================================
    knifeSharpeningTimeMS        : INT := 5000;    // [ms] Sharpening pulse time / Tempo de afiação


    knifeLubrificationTimeMS     : INT := 1;    // [ms] Lubrication pulse time / Tempo de lubrificação

	
	homeStartNextAxisDelay		: TIME := T#5S;	
		
	
	
    // ------------------------------------------------------------
    // Offsets
    // ------------------------------------------------------------
    knifeOffsetArr : ARRAY [1..20] OF REAL :=
        [-2, -1, 0, 3.5, 1.8, 0, 0, 0, 0, 0, 0, 0, 0, 0, 0, 0, 0, 0, 0, 0];

    scorerOffsetArr : ARRAY [1..20] OF REAL :=
        [5, -3, 4, -3, -3, 54, -6, 6, 0, 0, 0, 0, 0, 0, 0, 0, 0, 0, 0, 0];

    scorerHeightArr : ARRAY [1..5] OF REAL := [1.0, 0.8, 0.5, 0.5, 0.5];

    // ------------------------------------------------------------
    // Limits (min/max)
    // ------------------------------------------------------------
    knifeMaxPostionArr : ARRAY [1..20] OF INT :=
        [1265, 1080, 1220, 1907, 2060, 0, 0, 0, 0, 0, 0, 0, 0, 0, 0, 0, 0, 0, 0, 0];

    knifeMinPostionArr : ARRAY [1..20] OF INT :=
        [184, 330, 477, 0, 0, 0, 0, 0, 0, 0, 0, 0, 0, 0, 0, 0, 0, 0, 0, 0];

    scorerMaxPostionArr : ARRAY [1..20] OF INT :=
        [968, 968, 1120, 1120, 1864, 1890, 2004, 2050, 0, 0, 0, 0, 0, 0, 0, 0, 0, 0, 0, 0];

    scorerMinPostionArr : ARRAY [1..20] OF INT :=
        [204, 202, 364, 340, 1060, 1130, 1220, 1269, 0, 0, 0, 0, 0, 0, 0, 0, 0, 0, 0, 0];

	
arrFlapPosition : ARRAY[1..27] OF INT := [
    880,   // 1  (50   + 830)
    975,   // 2  (145  + 830)
    1065,  // 3  (235  + 830)
    1165,  // 4  (335  + 830)
    1255,  // 5  (425  + 830)
    1350,  // 6  (520  + 830)
    1445,  // 7  (615  + 830)
    1535,  // 8  (705  + 830)
    1630,  // 9  (800  + 830)
    1725,  // 10 (895  + 830)
    1815,  // 11 (985  + 830)
    1910,  // 12 (1080 + 830)
    2005,  // 13 (1175 + 830)
    2095,  // 14 (1265 + 830)
    2185,  // 15 (1355 + 830)
    2280,  // 16 (1450 + 830)
    2375,  // 17 (1545 + 830)
    2470,  // 18 (1640 + 830)
    2560,  // 19 (1730 + 830)
    2655,  // 20 (1825 + 830)
    2750,  // 21 (1920 + 830)
    2840,  // 22 (2010 + 830)
    2935,  // 23 (2105 + 830)
    3030,  // 24 (2200 + 830)
    3125,  // 25 (2295 + 830)
    3215,  // 26 (2385 + 830)
    3315   // 27 (2485 + 830)
];


minLineSpeed		: REAL := 20.0;
knifeSpeedOffset	: REAL := 2;
scorerSpeedOffset	: REAL := 1.05;
		




	
    fluteNameArr  : ARRAY [1..5] OF STRING := [ 'B', 'C', 'BC', 'E', '' ];




    //=================================================================
    // HOME POSITIONS (REFERENCE / ZERO)
    //=================================================================
    // NOTE: Define the mechanical reference position for each tool side.
    knifeOperatorSideHomePosition        : LREAL := 1947.5; // Knife home OS / Home faca lado operador
    knifeDriveSideHomePosition           : LREAL := 2247.5; // Knife home DS / Home faca lado acionamento

    upperScorerOperatorSideHomePosition  : LREAL:= 1947.5; // Upper scorer home OS / Home vinco superior lado operador
    upperScorerDriveSideHomePosition     : LREAL:= 2247.5; // Upper scorer home DS / Home vinco superior lado acionamento

    lowerScorerOperatorSideHomePosition  : LREAL:= 1947.5; // Lower scorer home OS / Home vinco inferior lado operador
    lowerScorerDriveSideHomePosition     : LREAL:= 2247.5; // Lower scorer home DS / Home vinco inferior lado acionamento

	
    knifeOperatorSideHomeSensorPosition        : LREAL := 883; // Knife home OS / Home faca lado operador
    knifeDriveSideHomeSensorPosition           : LREAL := 3275 ; // Knife home DS / Home faca lado acionamento

    upperScorerOperatorSideHomeSensorPosition  : LREAL:= 847; // Upper scorer home OS / Home vinco superior lado operador
    upperScorerDriveSideHomeSensorPosition     : LREAL:= 3433; // Upper scorer home DS / Home vinco superior lado acionamento

    lowerScorerOperatorSideHomeSensorPosition  : LREAL:= 761; // Lower scorer home OS / Home vinco inferior lado operador
    lowerScorerDriveSideHomeSensorPosition     : LREAL:= 3344; // Lower scorer home DS / Home vinco inferior lado acionamento
	
	
	

    knifeOperatorSideParkingPosition          : INT;  // Knife park OS / Estacionamento faca lado operador
    knifeDriveSideParkingPosition             : INT;  // Knife park DS / Estacionamento faca lado acionamento

    upperScorerOperatorSideParkingPosition    : INT;  // Upper scorer park OS / Estacionamento vinco superior lado operador
    upperScorerDriveSideParkingPosition       : INT;  // Upper scorer park DS / Estacionamento vinco superior lado acionamento

    lowerScorerOperatorSideParkingPosition    : INT;  // Lower scorer park OS / Estacionamento vinco inferior lado operador
    lowerScorerDriveSideParkingPosition       : INT;  // Lower scorer park DS / Estacionamento vinco inferior lado acionamento

    //=================================================================
    // MOTION PROFILES (POSITIONING / GENERAL / MANUAL)
    //=================================================================
	
	knifeMinDistance : LREAL := 150.0;
	scorerMinDistance : LREAL := 95.0;
	
	
	

    // Manual jog motion (HMI / maintenance)
    toolJogMotionVelocity     : LREAL := 10.0;    // [mm/s] Manual speed / Velocidade manual
    toolJogMotionAccel        : LREAL := 9214.76; // [mm/s²] Manual accel / Aceleração manual
    toolJogMotionDecel        : LREAL := 9214.76; // [mm/s²] Manual decel / Desaceleração manual
    toolJogMotionJerk         : LREAL := 276443; // [mm/s³] Manual jerk / Jerk manual
	


	

    //=================================================================
    // TOOL OFFSETS / CALIBRATION ARRAYS
    //=================================================================
    // Offsets are typically used to compensate mechanical differences per tool.
    // Keep array size >= maximum possible tools (configured by machineNumberOf*).
    knifePositionCorrectionArr  	: ARRAY [1..20] OF REAL := [ 00.0, 00.0, 00.0, 00.0,  00.0, 00.0,  00.0,  00.0,  00.0,  00.0, 00.0,  00.0,  00.0,  00.0,  00.0,  00.0,  00.0,  00.0,  00.0,  00.0 ];
    scorerPositionCorrectionArr  	: ARRAY [1..20] OF REAL := [ 00.0, 00.0, 00.0, 00.0,  00.0, 00.0,  00.0,  00.0,  00.0,  00.0, 00.0,  00.0,  00.0,  00.0,  00.0,  00.0,  00.0,  00.0,  00.0,  00.0 ];
    scorerAlignmentCompensationArr  : ARRAY [1..20] OF REAL := [ 00.0, 00.0, 00.0, 00.0,  00.0, 00.0,  00.0,  00.0,  00.0,  00.0, 00.0,  00.0,  00.0,  00.0,  00.0,  00.0,  00.0,  00.0,  00.0,  00.0 ];

dsTrimDuctHomeSensorPosition : REAL;
scorerHeightSensorPosition : REAL;




















		
END_STRUCT
END_TYPE

// ---- Library/Machine/Slitter/DataTypes/Hmi/slitterStatus_TypeStruct.TcDUT
TYPE slitterStatus_TypeStruct :
STRUCT



//	sharpeningSolenoidArr			: ARRAY [1..20] OF BOOL;	(*Sharpening solenoid output*)
//	lubrificationSolenoidArr		: ARRAY [1..20] OF BOOL;	(*Lubrificaion solenoid output*)
//	knifeRunningMetersArr			: ARRAY [1..20] OF INT;		(*Knife running meters until sharpening*)
//	lubrificationRunningMetersArr	: ARRAY [1..20] OF INT;		(*Knife running meters until lubrificaion*)
//	knifeRunningMetersTotalArr		: ARRAY [1..20] OF DINT;	(*Knife total running meters without blade change*)

	doubleFacerSpeed				: INT;

	positioningRunning				: BOOL;						(*Positioning running*)
	positioningFinished				: BOOL;						(*Positioning finished*)
	
	slitterCutting					: BOOL;						(*Slitter cutting the material (At least one knife enabled)*)
	
	
	knifeMotorRunning				: BOOL;
	knifeMotorSpeedRPM				: INT;
	knifeMotorSpeedMPM				: INT;
	knifeMotorCurrent				: INT;

	scorerMotorRunning				: BOOL;
	scorerMotorSpeedRPM				: INT;
	scorerMotorSpeedMPM				: INT;
	scorerMotorCurrent				: INT;

	knifeAxisSpeed					: LREAL;
	knifeAxisPosition				: DINT;
	knifeAxisState					: STRING;

	innerScorerAxisSpeed			: LREAL;	
	innerScorerAxisPosition			: DINT;
	innerScorerAxisState			: STRING;
	
	outerScorerAxisSpeed			: LREAL;		
	outerScorerAxisPosition			: DINT;
	outerScorerAxisState			: STRING;

	scorerHeight					: REAL;	(*Scorer actual height in milimiters*)
	alarmActive						: BOOL;	(**)
	

    // ─────────────── TOOL POSITIONS ───────────────
    knifePosition                    : ARRAY [1..7] OF REAL;   // Knife actual position (machine units, e.g. mm)
    scorerPosition                   : ARRAY [1..12] OF REAL;  // Scorer actual position (machine units, e.g. mm)

    // ─────────────── FLAPS / DIVERTERS ───────────────
    flapSolenoidArr                  : ARRAY [1..27] OF BOOL;  // Flap solenoid output command/status (per flap)

	
    // ─────────────── KNIFE SERVICE / MAINTENANCE STATUS ───────────────
    sharpeningSolenoidArr            : ARRAY [1..7] OF BOOL;   // Sharpening solenoid output command/status (per knife)
    lubrificationSolenoidArr         : ARRAY [1..7] OF BOOL;   // Lubrication solenoid output command/status (per knife)

    knifeRunningMetersArr            : ARRAY [1..7] OF INT;    // Running meters since last sharpening (per knife)
    lubrificationRunningMetersArr    : ARRAY [1..7] OF INT;    // Running meters since last lubrication (per knife)
    knifeRunningMetersTotalArr       : ARRAY [1..7] OF DINT;   // Total running meters since last blade change (per knife)
	
	

END_STRUCT
END_TYPE

// ---- Library/Machine/Stacker/Simple/DataTypes/hmiAlarmsSimpleStacker_TypeStruct.TcDUT
TYPE hmiAlarmsSimpleStacker_TypeStruct :
STRUCT

    //==============================================================
    // General / system alarms
    //==============================================================
    safetyCircuitNotOk                 : BOOL;
    systemFaultActive                  : BOOL;
    systemNotEnabled                   : BOOL;

    // EN: Generic safety feedback diagnostic alarms.
    // PT: Alarmes genéricos de diagnóstico dos retornos de segurança.
    safetyFeedback1NotOk               : BOOL;
    safetyFeedback2NotOk               : BOOL;
    safetyFeedback3NotOk               : BOOL;
    safetyFeedback4NotOk               : BOOL;
    safetyFeedback5NotOk               : BOOL;
    safetyFeedback6NotOk               : BOOL;
    safetyFeedback7NotOk               : BOOL;
    safetyFeedback8NotOk               : BOOL;

    //==============================================================
    // Sheet conveyor group alarms
    //==============================================================
    sheetConveyor1DriveNotOk           : BOOL;
    sheetConveyor2DriveNotOk           : BOOL;
    sheetConveyor3DriveNotOk           : BOOL;
    sheetConveyorGroupFault            : BOOL;
    synchronizedConveyorsNotRunning    : BOOL;

    //==============================================================
    // Sheet stack separation alarms / indications
    //==============================================================
    sheetStackSeparationNotReady       : BOOL;
    sheetStackSeparationActive         : BOOL;
    sheetStackBrakeActive              : BOOL;

    //==============================================================
    // Sheet stack discharge sequence alarms / indications
    //==============================================================
    sheetStackDischargeFault           : BOOL;
    sheetStackDischargeLastCycleNotOk  : BOOL;
    sheetStackDischargeTimeout         : BOOL;
    sheetStackDischargeManualSkip      : BOOL;

    //==============================================================
    // Sheet stack discharge conveyor alarms
    //==============================================================
    sheetStackDischargeConveyorDriveNotOk : BOOL;
    sheetStackDischargeConveyorFault      : BOOL;

    //==============================================================
    // Backstop alarms / indications
    //==============================================================
    backstopDriveNotOk                 : BOOL;
    backstopFault                      : BOOL;
    backstopNotHomed                   : BOOL;
    backstopNotInPosition              : BOOL;

    backstopSafeMaxLimitActive         : BOOL;
    backstopSafeMinLimitActive         : BOOL;
    backstopMaxLimitActive             : BOOL;
    backstopMinLimitActive             : BOOL;

    backstopManualInterventionActive   : BOOL;

    //==============================================================
    // Conveyor leveler alarms / indications
    //==============================================================
    conveyorLevelerDriveNotOk          : BOOL;
    conveyorLevelerFault               : BOOL;
    conveyorLevelerNotHomed            : BOOL;
    conveyorLevelerNotInPosition       : BOOL;

    conveyorLevelerUpperSafetyLimitActive : BOOL;
    conveyorLevelerLowerSafetyLimitActive : BOOL;
    conveyorLevelerUpperLimitActive       : BOOL;
    conveyorLevelerLowerLimitActive       : BOOL;

END_STRUCT
END_TYPE

// ---- Library/Machine/Stacker/Simple/DataTypes/hmiCommandsSimpleStacker_TypeStruct.TcDUT

TYPE hmiCommandsSimpleStacker_TypeStruct :
STRUCT

    //==============================================================
    // System master commands
    //==============================================================
    startCmd                                : BOOL; // EN: Master start command
    stopCmd                                 : BOOL; // EN: Master stop command
    resetCmd                                : BOOL; // EN: Fault reset command


    //==============================================================
    // Sheet conveyor group commands
    //==============================================================
    sheetConveyorsSpeedUpCmd                : BOOL; // EN: Momentary speed-up command for sheet conveyors


    //==============================================================
    // Sheet handling commands
    //==============================================================
    packageCompleteCmd                      : BOOL; // EN: Package complete / discharge cycle request
    sheetDiscardCmd                         : BOOL; // EN: Sheet discard command
    noCrushRollersUpCmd                     : BOOL; // EN: No-crush rollers up command


    //==============================================================
    // Backstop commands
    //==============================================================
    backstopAutoCmd                         : BOOL; // EN: Enables backstop automatic mode
    backstopHomeCmd                         : BOOL; // EN: Manual backstop homing command
    backstopExecutePositioningCmd           : BOOL; // EN: Execute programmed backstop positioning

    backstopOpenCmd                         : BOOL; // EN: Manual backstop open command
    backstopCloseCmd                        : BOOL; // EN: Manual backstop close command


    //==============================================================
    // Conveyor leveler commands
    //==============================================================
    conveyorLevelerAutoCmd                  : BOOL; // EN: Enables conveyor leveler automatic mode
    conveyorLevelerHomeCmd                  : BOOL; // EN: Manual conveyor leveler homing command

    conveyorLevelerUpCmd                    : BOOL; // EN: Manual conveyor leveler up command
    conveyorLevelerDownCmd                  : BOOL; // EN: Manual conveyor leveler down command


    //==============================================================
    // Sheet stack discharge conveyor commands
    //==============================================================
    sheetStackDischargeConveyorManualRunCmd : BOOL; // EN: Momentary manual run command for discharge conveyor

END_STRUCT
END_TYPE

// ---- Library/Machine/Stacker/Simple/DataTypes/hmiStatusSimpleStacker_TypeStruct.TcDUT
TYPE hmiStatusSimpleStacker_TypeStruct :
STRUCT

    //==============================================================
    // System general status
    //==============================================================
    systemRunEnable                         : BOOL;        // EN: Master system run enable
    safetyCircuitOk                         : BOOL;        // EN: Safety circuit status
    faultActive                             : BOOL;        // EN: General fault active
    deviceState                             : STRING(30);  // EN: General device state text


    //==============================================================
    // Sheet conveyor group status
    //==============================================================
    synchronizedConveyorsRunning            : BOOL;        // EN: All synchronized conveyors running

    sheetConveyor1Run                       : BOOL;        // EN: Sheet conveyor 1 run output
    sheetConveyor2Run                       : BOOL;        // EN: Sheet conveyor 2 run output
    sheetConveyor3Run                       : BOOL;        // EN: Sheet conveyor 3 run output

    sheetConveyor1SpeedRefMPM               : REAL;        // EN: Sheet conveyor 1 speed reference [m/min]
    sheetConveyor2SpeedRefMPM               : REAL;        // EN: Sheet conveyor 2 speed reference [m/min]
    sheetConveyor3SpeedRefMPM               : REAL;        // EN: Sheet conveyor 3 speed reference [m/min]

    syncConveyorsState                      : INT;         // EN: Synchronized conveyor group state code


    //==============================================================
    // Sheet stack separation status
    //==============================================================
    sheetStackSeparationReady               : BOOL;        // EN: Stack separation ready
    sheetStackSeparationActive              : BOOL;        // EN: Stack separation active
    sheetStackBrakeActive                   : BOOL;        // EN: Stack brake active

    sheetStackSeparationDistanceM           : REAL;        // EN: Current separation distance [m]
    sheetStackSeparationTargetDistanceM     : REAL;        // EN: Target separation distance [m]


    //==============================================================
    // Sheet stack discharge sequence status
    //==============================================================
    sheetStackDischargeState                : STRING(30);  // EN: Discharge sequence state text
    sheetStackDischargeStateCode            : INT;         // EN: Discharge sequence state code

    sheetStackDischargePending              : BOOL;        // EN: Discharge cycle pending
    sheetStackDischargeActive               : BOOL;        // EN: Discharge cycle active
    sheetStackDischargeStarted              : BOOL;        // EN: Discharge cycle started pulse/status
    sheetStackDischargeFinished             : BOOL;        // EN: Discharge cycle finished pulse/status

    sheetStackDischargeFault                : BOOL;        // EN: Discharge sequence fault
    sheetStackDischargeFaultCode            : INT;         // EN: Current discharge fault code

    sheetStackDischargeLastCycleOk          : BOOL;        // EN: Last discharge cycle completed successfully
    sheetStackDischargeLastResultCode       : INT;         // EN: Last discharge result code
    sheetStackDischargeLastFaultStepCode    : INT;         // EN: Last discharge fault step code
    sheetStackDischargeLastFaultCode        : INT;         // EN: Last discharge fault code


    //==============================================================
    // Sheet stack discharge conveyor status
    //==============================================================
    sheetStackDischargeConveyorState        : STRING(30);  // EN: Discharge conveyor state text
    sheetStackDischargeConveyorRun          : BOOL;        // EN: Discharge conveyor run output
    sheetStackDischargeConveyorSpeedRefMPM  : REAL;        // EN: Discharge conveyor speed reference [m/min]

    sheetStackDischargeConveyorFault        : BOOL;        // EN: Discharge conveyor fault
    sheetStackDischargeConveyorFaultCode    : INT;         // EN: Discharge conveyor fault code


    //==============================================================
    // Backstop status
    //==============================================================
    backstopState                           : STRING(30);  // EN: Backstop state text
    backstopHomed                           : BOOL;        // EN: Backstop homing completed
    backstopHomeRunning                     : BOOL;        // EN: Backstop homing sequence running
    backstopInPosition                      : BOOL;        // EN: Backstop is inside target tolerance

    backstopPositionMm                      : REAL;        // EN: Actual backstop position [mm]
    backstopTargetPositionMm                : REAL;        // EN: Active backstop target position [mm]
    backstopPositionErrorMm                 : REAL;        // EN: Backstop position error [mm]

    backstopRunFw                           : BOOL;        // EN: Backstop forward/open run output
    backstopRunRev                          : BOOL;        // EN: Backstop reverse/close run output
    backstopSpeedRefMmps                    : REAL;        // EN: Backstop speed reference [mm/s]

    backstopPlateUpSolenoid                 : BOOL;        // EN: Backstop plate up solenoid
    backstopSetEncoderPosition              : BOOL;        // EN: Backstop set encoder pulse
    backstopSetEncoderPositionMm            : REAL;        // EN: Backstop set encoder position [mm]

    backstopManualInterventionActive        : BOOL;        // EN: Manual intervention memory active
    backstopManualInterventionPositionMm    : REAL;        // EN: Stored manual intervention position [mm]

    backstopFault                           : BOOL;        // EN: Backstop fault
    backstopFaultCode                       : INT;         // EN: Backstop fault code


    //==============================================================
    // Conveyor leveler status
    //==============================================================
    conveyorLevelerState                    : STRING(30);  // EN: Conveyor leveler state text
    conveyorLevelerHomed                    : BOOL;        // EN: Conveyor leveler homing completed
    conveyorLevelerInPosition               : BOOL;        // EN: Conveyor leveler is inside target tolerance

    conveyorLevelerPositionMm               : REAL;        // EN: Actual conveyor leveler position [mm]
    conveyorLevelerTargetPositionMm         : REAL;        // EN: Active conveyor leveler target position [mm]
    conveyorLevelerPositionErrorMm          : REAL;        // EN: Conveyor leveler position error [mm]

    conveyorLevelerRunUp                    : BOOL;        // EN: Conveyor leveler up run output
    conveyorLevelerRunDown                  : BOOL;        // EN: Conveyor leveler down run output
    conveyorLevelerBrakeRelease             : BOOL;        // EN: Conveyor leveler brake release output
    conveyorLevelerSpeedRefMmps             : REAL;        // EN: Conveyor leveler speed reference [mm/s]

    conveyorLevelerSetEncoderPosition       : BOOL;        // EN: Conveyor leveler set encoder pulse
    conveyorLevelerSetEncoderPositionMm     : REAL;        // EN: Conveyor leveler set encoder position [mm]

    conveyorLevelerFault                    : BOOL;        // EN: Conveyor leveler fault
    conveyorLevelerFaultCode                : INT;         // EN: Conveyor leveler fault code


    //==============================================================
    // Process values
    //==============================================================
    lineSpeedMPM                            : REAL;        // EN: Current line speed [m/min]
    sheetLengthMm                           : REAL;        // EN: Current sheet length [mm]
    stackHeightMm                           : REAL;        // EN: Current stack height [mm]


    //==============================================================
    // Input / drive status mirror
    //==============================================================
    sheetConveyor1DriveOk                   : BOOL;        // EN: Sheet conveyor 1 drive OK
    sheetConveyor2DriveOk                   : BOOL;        // EN: Sheet conveyor 2 drive OK
    sheetConveyor3DriveOk                   : BOOL;        // EN: Sheet conveyor 3 drive OK

    backstopDriveOk                         : BOOL;        // EN: Backstop drive OK
    conveyorLevelerDriveOk                  : BOOL;        // EN: Conveyor leveler drive OK
    sheetStackDischargeConveyorDriveOk      : BOOL;        // EN: Discharge conveyor drive OK

END_STRUCT
END_TYPE

// ---- Library/Machine/Stacker/Cpx/DataTypes/ComplexStackerConfig_TypeStruct.TcDUT
TYPE ComplexStackerConfig_TypeStruct :
STRUCT

    //=================================================================
    // 01 - General line / stacker speed configuration
    //=================================================================

    // EN: Normal stacker speed ratio relative to line speed.
    //     Example: 0.17 = stacker runs at 17% of line speed.
    // PT: Fator normal de velocidade do stacker em relação à velocidade da linha.
    //     Exemplo: 0.17 = stacker trabalha com 17% da velocidade da linha.
    stackerSpeedRatio                         : REAL := 0.17;

    // EN: Minimum and maximum speed reference allowed for sheet conveyors [m/min].
    // PT: Referência mínima e máxima permitida para as esteiras de chapas [m/min].
    minimumSpeedMPM                           : REAL := 10.0;
    maximumSpeedMPM                           : REAL := 80.0;

    // EN: Maximum ramp velocity for conveyor speed references [m/min/s].
    // PT: Velocidade máxima da rampa para referências das esteiras [m/min/s].
    rampVelocityUpMaxMPMps                    : REAL := 1000.0;
    rampVelocityDownMaxMPMps                  : REAL := 1000.0;

    // EN: Ramp acceleration / deceleration used by S-ramp smoothing [m/min/s²].
    // PT: Aceleração / desaceleração usada na suavização da rampa S [m/min/s²].
    rampAccelerationUpMPMps2                  : REAL := 1000.0;
    rampAccelerationDownMPMps2                : REAL := 1000.0;


    //=================================================================
    // 02 - Sheet conveyor group: speed trim and mechanical length
    //=================================================================

    // EN: Individual speed trim for each synchronized sheet conveyor.
    //     1.0 = no correction.
    // PT: Correção individual de velocidade para cada esteira sincronizada.
    //     1.0 = sem correção.
    sheetConveyor1SpeedTrim                   : REAL := 1.0;
    sheetConveyor2SpeedTrim                   : REAL := 1.0;
    sheetConveyor3SpeedTrim                   : REAL := 1.0;
    sheetConveyor4SpeedTrim                   : REAL := 1.0;

    // EN: Sheet conveyor mechanical length [m].
    // PT: Comprimento mecânico da esteira de chapas [m].
    sheetConveyor1LengthM                     : REAL := 1.85;
    sheetConveyor2LengthM                     : REAL := 1.0;
    sheetConveyor3LengthM                     : REAL := 2.0;
    sheetConveyor4LengthM                     : REAL := 2.0;

    // EN: Additional speed reference applied to sheet conveyors 1, 2 and 3
    //     when the external speed-up command is active [m/min].
    // PT: Referência adicional aplicada nas esteiras 1, 2 e 3
    //     quando o comando externo de aceleração estiver ativo [m/min].
    sheetConveyorsSpeedUpMPM                  : REAL := 20.0;


    //=================================================================
    // 03 - Sheet conveyor group: package separation
    //=================================================================

    // EN: Speed multiplier used during package separation.
    //     Example: 1.50 = 50% faster than normal speed.
    // PT: Multiplicador de velocidade usado durante a separação de pacote.
    //     Exemplo: 1.50 = 50% acima da velocidade normal.
    packageGapSpeedRatio                      : REAL := 3.0;

    // EN: Additional fixed speed offset during package separation [m/min].
    // PT: Offset fixo adicional de velocidade durante a separação de pacote [m/min].
    packageGapSpeedOffsetMPM                  : REAL := 0.0;

    // EN: Minimum line speed used as the conveyor speed calculation reference
    //     while package separation is active [m/min].
    //     Set to 0.0 to keep the actual line speed without a discharge override.
    // PT: Velocidade mínima da linha usada como referência para o cálculo das
    //     esteiras enquanto a separação da pilha estiver ativa [m/min].
    //     Usar 0.0 para manter a velocidade real da linha sem sobreposição no descarte.
    packageDischargeLineSpeedThresholdMPM     : REAL := 0.0;

    // EN: Minimum valid differential speed used for separation tracking [m/min].
    // PT: Velocidade diferencial mínima válida usada no rastreamento da separação [m/min].
    minimumOpeningSpeedMPM                    : REAL := 1.0;


    //=================================================================
    // 04 - Elevator: speed trim and position limits
    //=================================================================

    // EN: Individual speed trim for elevator synchronized movement.
    //     1.0 = no correction.
    // PT: Correção individual de velocidade para movimento sincronizado do elevador.
    //     1.0 = sem correção.
    elevatorSpeedTrim                  : REAL := 1.0;

    // EN: Minimum and maximum allowed elevator position [mm].
    // PT: Posição mínima e máxima permitida para o elevador [mm].
    elevatorMinPositionMm              : REAL := 10.0;
    elevatorMaxPositionMm              : REAL := 150.0;


    //=================================================================
    // 05 - Elevator: automatic positioning
    //=================================================================

    // EN: Offset added to stack height to calculate elevator target [mm].
    // PT: Offset somado à altura da pilha para calcular o alvo do elevador [mm].
    elevatorStackHeightOffsetMm        : REAL := 0.0;

    // EN: Position tolerance to consider elevator in position [mm].
    // PT: Tolerância de posição para considerar o elevador em posição [mm].
    elevatorPositionToleranceMm        : REAL := 2.0;

    // EN: Proportional gain for elevator position control [(mm/s)/mm].
    // PT: Ganho proporcional do controle de posição do elevador [(mm/s)/mm].
    elevatorPositionKp                 : REAL := 5.0;

    // EN: Maximum upward speed for proportional automatic positioning [mm/s].
    // PT: Velocidade máxima de subida no posicionamento automático proporcional [mm/s].
    elevatorAutomaticUpSpeedMmps       : REAL := 30.0;

    // EN: Maximum downward speed for proportional automatic positioning [mm/s].
    // PT: Velocidade máxima de descida no posicionamento automático proporcional [mm/s].
    elevatorAutomaticDownSpeedMmps     : REAL := 30.0;

    //=================================================================
    // 06 - Elevator: manual movement
    //=================================================================

    // EN: Manual up/down speed for elevator [mm/s].
    // PT: Velocidade manual para subir/descer o elevador [mm/s].
    elevatorManualSpeedMmps            : REAL := 50.0;

    // EN: Distance from each configured endpoint where manual movement
    //     changes to reduced speed [mm].
    // PT: Distância a partir de cada extremidade configurada onde o movimento
    //     manual passa para velocidade reduzida [mm].
    elevatorManualLowSpeedZoneMm       : REAL := 300.0;

    // EN: Manual speed multiplier inside the low-speed zone [0.0..1.0].
    // PT: Multiplicador da velocidade manual dentro da zona lenta [0.0..1.0].
    elevatorManualLowSpeedFactor       : REAL := 0.3;

    // EN: First downward speed while the stack level sensor is active [mm/s].
    // PT: Primeira velocidade de descida enquanto o sensor de nível estiver acionado [mm/s].
    elevatorLevelingSpeed1Mmps         : REAL := 5.0;

    // EN: Second downward speed when the stack level sensor remains active [mm/s].
    // PT: Segunda velocidade de descida quando o sensor de nível permanecer acionado [mm/s].
    elevatorLevelingSpeed2Mmps         : REAL := 15.0;

    // EN: Time before changing from leveling speed 1 to speed 2.
    // PT: Tempo antes de mudar da velocidade 1 para a velocidade 2 de nivelamento.
    elevatorLevelingSpeed2Delay        : TIME := T#2S;


    //=================================================================
    // 07 - Elevator: homing and encoder set
    //=================================================================

    // EN: Elevator homing speed [mm/s].
    // PT: Velocidade de homing do elevador [mm/s].
    elevatorHomingSpeedMmps            : REAL := 30.0;

    // EN: Slow upward speed used to leave the lower home sensor [mm/s].
    // PT: Velocidade lenta de subida usada para liberar o sensor inferior de home [mm/s].
    elevatorHomingReleaseSpeedMmps     : REAL := 5.0;

    // EN: Maximum allowed time for elevator homing movement.
    // PT: Tempo máximo permitido para o movimento de homing do elevador.
    elevatorHomingTimeout              : TIME := T#30S;

    // EN: Pulse time for elevator encoder position set command.
    // PT: Tempo do pulso para comando de set da posição do encoder do elevador.
    elevatorSetEncoderPulseTime        : TIME := T#200MS;

    // EN: Stabilization time after leaving the lower home sensor.
    // PT: Tempo de estabilização após liberar o sensor inferior de home.
    elevatorHomeSettleDelay            : TIME := T#500MS;

    // EN: Encoder position applied after the lower home sensor is released [mm].
    // PT: Posição aplicada ao encoder após liberar o sensor inferior de home [mm].
    elevatorHomePositionMm             : REAL := 10.0;


    //=================================================================
    // 08 - Elevator: magnetic brake
    //=================================================================

    // EN: Delay between brake release command and motor movement permission.
    // PT: Atraso entre o comando de liberação do freio e a permissão de movimento do motor.
    elevatorBrakeReleaseDelay          : TIME := T#300MS;

    // EN: Time to keep the brake released after movement stops.
    // PT: Tempo para manter o freio liberado após a parada do movimento.
    elevatorBrakeHoldTime              : TIME := T#2S;

    //=================================================================
    // 09 - Backstop: position limits
    //=================================================================

    // EN: Minimum and maximum allowed backstop position [mm].
    // PT: Posição mínima e máxima permitida para o backstop [mm].
    backstopMinPositionMm                     : REAL := 300.0;
    backstopMaxPositionMm                     : REAL := 5000.0;


    //=================================================================
    // 10 - Backstop: homing and encoder set
    //=================================================================

    // EN: Homing direction. -1 = close/min limit, +1 = open/max limit.
    // PT: Direção de homing. -1 = fechar/limite mínimo, +1 = abrir/limite máximo.
    backstopHomeDirection                     : INT := 1;

    // EN: Encoder position value to set after homing is completed [mm].
    // PT: Valor de posição gravado no encoder após finalizar o homing [mm].
    backstopHomePositionMm                    : REAL := 2985.0;

    // EN: Backstop homing speed [mm/s].
    // PT: Velocidade de homing do backstop [mm/s].
    backstopHomingSpeedMmps                   : REAL := 150.0;

    // EN: Maximum allowed time for backstop homing movement.
    // PT: Tempo máximo permitido para o movimento de homing do backstop.
    backstopHomingTimeout                     : TIME := T#40S;

    // EN: Pulse time for backstop encoder position set command.
    // PT: Tempo do pulso para comando de set da posição do encoder do backstop.
    backstopSetEncoderPulseTime               : TIME := T#200MS;


    //=================================================================
    // 11 - Backstop: automatic positioning
    //=================================================================

    // EN: Offset added to sheet length to calculate automatic backstop target [mm].
    // PT: Offset somado ao comprimento da chapa para calcular o alvo automático do backstop [mm].
    backstopSheetLengthOffsetMm               : REAL := 0.0;

    // EN: Position tolerance to consider the backstop in position [mm].
    // PT: Tolerância de posição para considerar o backstop em posição [mm].
    backstopPositionToleranceMm               : REAL := 5.0;

    // EN: Proportional gain for backstop position control [(mm/s)/mm].
    // PT: Ganho proporcional do controle de posição do backstop [(mm/s)/mm].
    backstopPositionKp                        : REAL := 3.0;

    // EN: Maximum speed allowed in automatic backstop positioning [mm/s].
    // PT: Velocidade máxima permitida no posicionamento automático do backstop [mm/s].
    backstopAutoMaxSpeedMmps                  : REAL := 400.0;

    // EN: Minimum movement speed when the position error is above tolerance [mm/s].
    // PT: Velocidade mínima de movimento quando o erro de posição estiver acima da tolerância [mm/s].
    backstopMinMoveSpeedMmps                  : REAL := 15.0;


    //=================================================================
    // 12 - Backstop: manual movement
    //=================================================================

    // EN: Manual open/close speed for backstop [mm/s].
    // PT: Velocidade manual para abrir/fechar o backstop [mm/s].
    backstopManualSpeedMmps                   : REAL := 80.0;

    // EN: Minimum speed reference required to enable backstop drive run [mm/s].
    // PT: Referência mínima de velocidade necessária para liberar RUN do acionamento do backstop [mm/s].
    backstopRunMinSpeedMmps                   : REAL := 10.0;


    //=================================================================
    // 13 - Sheet stack discharge conveyor
    //=================================================================

    // EN: Sheet stack discharge conveyor speed reference [m/min].
    // PT: Referência de velocidade da esteira de descarga da pilha [m/min].
    sheetStackDischargeConveyorSpeedMPM       : REAL := 70.0;

    // EN: Minimum running time for the sheet stack discharge conveyor.
    // PT: Tempo mínimo de giro da esteira de descarga da pilha.
    sheetStackDischargeTime                   : TIME := T#2S;

    // EN: Maximum time allowed to confirm that the elevator platform is clear.
    // PT: Tempo máximo permitido para confirmar que a plataforma do elevador está livre.
    sheetStackDischargePlatformClearTimeout   : TIME := T#30S;


    //=================================================================
    // 14 - Sheet stack discharge sequence: backstop movement
    //=================================================================

    // EN: Additional backstop opening during sheet stack discharge [mm].
    // PT: Abertura adicional do backstop durante a descarga da pilha [mm].
    backstopDischargeOpenOffsetMm             : REAL := 100.0;


    //=================================================================
    // 15 - Sheet stack discharge sequence: step timeouts
    //=================================================================

    // EN: Maximum time to wait for package separation before discharge sequence continues.
    // PT: Tempo máximo de espera pela separação do pacote antes da sequência de descarga continuar.
    sheetStackDischargeWaitSeparationTimeout  : TIME := T#10S;

    // EN: Maximum time allowed for discharge positioning movement.
    // PT: Tempo máximo permitido para o movimento de posicionamento da descarga.
    sheetStackDischargePositioningTimeout     : TIME := T#10S;

    // EN: Maximum time allowed to confirm/start discharge conveyor movement.
    // PT: Tempo máximo permitido para confirmar/iniciar o movimento da esteira de descarga.
    sheetStackDischargeConveyorStartTimeout   : TIME := T#3S;

    // EN: Maximum time allowed for backstop return movement after discharge.
    // PT: Tempo máximo permitido para o retorno do backstop após a descarga.
    sheetStackDischargeReturnTimeout          : TIME := T#10S;


